(* Logix 5000 project; controller reports 1756-L63 rev 20.15; software revision 20.04; part 20 of 52 *)

        [1198].log_data[8].valid := 1, [1198].log_data[9].valid := 1, [1198].log_data[10].valid := 1, [1198].log_data[11].valid := 1, [1198].log_data[12].valid := 1, [1198].log_data[13].valid := 1, [1198].log_data[14].valid := 1, [1198].log_data[15].valid := 1, [1198].log_data[16].valid := 1, [1198].log_data[17].valid := 1, [1198].log_data[18].valid := 1, [1198].log_data[19].valid := 1, [1198].time.Year := 2023, [1198].time.Month := 1, [1198].time.Day := 13, [1198].time.Hour := 20, [1198].time.Minute := 14, [1198].time.Second := 59, [1199].log_data[0].min := 1.0, [1199].log_data[0].max := 1.0, [1199].log_data[0].total := 300.0, [1199].log_data[0].time := 300.0, [1199].log_data[0].minminute := 15, [1199].log_data[0].maxminute := 15, [1199].log_data[0].valid := 1, [1199].log_data[1].valid := 1, [1199].log_data[2].valid := 1, [1199].log_data[3].valid := 1, [1199].log_data[4].valid := 1, [1199].log_data[5].valid := 1, [1199].log_data[6].valid := 1, [1199].log_data[7].valid := 1, [1199].log_data[8].valid := 1, [1199].log_data[9].valid := 1, [1199].log_data[10].valid := 1, [1199].log_data[11].valid := 1, [1199].log_data[12].valid := 1, [1199].log_data[13].valid := 1, [1199].log_data[14].valid := 1, [1199].log_data[15].valid := 1, [1199].log_data[16].valid := 1, [1199].log_data[17].valid := 1, [1199].log_data[18].valid := 1, [1199].log_data[19].valid := 1, [1199].time.Year := 2023, [1199].time.Month := 1, [1199].time.Day := 13, [1199].time.Hour := 20, [1199].time.Minute := 19, [1199].time.Second := 59, [1200].log_data[0].min := 1.0, [1200].log_data[0].max := 1.0, [1200].log_data[0].total := 300.0, [1200].log_data[0].time := 300.0, [1200].log_data[0].minminute := 20, [1200].log_data[0].maxminute := 20, [1200].log_data[0].valid := 1, [1200].log_data[1].valid := 1, [1200].log_data[2].valid := 1, [1200].log_data[3].valid := 1,
        [1200].log_data[4].valid := 1, [1200].log_data[5].valid := 1, [1200].log_data[6].valid := 1, [1200].log_data[7].valid := 1, [1200].log_data[8].valid := 1, [1200].log_data[9].valid := 1, [1200].log_data[10].valid := 1, [1200].log_data[11].valid := 1, [1200].log_data[12].valid := 1, [1200].log_data[13].valid := 1, [1200].log_data[14].valid := 1, [1200].log_data[15].valid := 1, [1200].log_data[16].valid := 1, [1200].log_data[17].valid := 1, [1200].log_data[18].valid := 1, [1200].log_data[19].valid := 1, [1200].time.Year := 2023, [1200].time.Month := 1, [1200].time.Day := 13, [1200].time.Hour := 20, [1200].time.Minute := 24, [1200].time.Second := 59, [1201].log_data[0].min := 1.0, [1201].log_data[0].max := 1.0, [1201].log_data[0].total := 300.0, [1201].log_data[0].time := 300.0, [1201].log_data[0].minminute := 25, [1201].log_data[0].maxminute := 25, [1201].log_data[0].valid := 1, [1201].log_data[1].valid := 1, [1201].log_data[2].valid := 1, [1201].log_data[3].valid := 1, [1201].log_data[4].valid := 1, [1201].log_data[5].valid := 1, [1201].log_data[6].valid := 1, [1201].log_data[7].valid := 1, [1201].log_data[8].valid := 1, [1201].log_data[9].valid := 1, [1201].log_data[10].valid := 1, [1201].log_data[11].valid := 1, [1201].log_data[12].valid := 1, [1201].log_data[13].valid := 1, [1201].log_data[14].valid := 1, [1201].log_data[15].valid := 1, [1201].log_data[16].valid := 1, [1201].log_data[17].valid := 1, [1201].log_data[18].valid := 1, [1201].log_data[19].valid := 1, [1201].time.Year := 2023, [1201].time.Month := 1, [1201].time.Day := 13, [1201].time.Hour := 20, [1201].time.Minute := 29, [1201].time.Second := 59, [1202].log_data[0].min := 1.0, [1202].log_data[0].max := 1.0, [1202].log_data[0].total := 300.0, [1202].log_data[0].time := 300.0, [1202].log_data[0].minminute := 30, [1202].log_data[0].maxminute := 30,
        [1202].log_data[0].valid := 1, [1202].log_data[1].valid := 1, [1202].log_data[2].valid := 1, [1202].log_data[3].valid := 1, [1202].log_data[4].valid := 1, [1202].log_data[5].valid := 1, [1202].log_data[6].valid := 1, [1202].log_data[7].valid := 1, [1202].log_data[8].valid := 1, [1202].log_data[9].valid := 1, [1202].log_data[10].valid := 1, [1202].log_data[11].valid := 1, [1202].log_data[12].valid := 1, [1202].log_data[13].valid := 1, [1202].log_data[14].valid := 1, [1202].log_data[15].valid := 1, [1202].log_data[16].valid := 1, [1202].log_data[17].valid := 1, [1202].log_data[18].valid := 1, [1202].log_data[19].valid := 1, [1202].time.Year := 2023, [1202].time.Month := 1, [1202].time.Day := 13, [1202].time.Hour := 20, [1202].time.Minute := 34, [1202].time.Second := 59, [1203].log_data[0].min := 1.0, [1203].log_data[0].max := 1.0, [1203].log_data[0].total := 300.0, [1203].log_data[0].time := 300.0, [1203].log_data[0].minminute := 35, [1203].log_data[0].maxminute := 35, [1203].log_data[0].valid := 1, [1203].log_data[1].valid := 1, [1203].log_data[2].valid := 1, [1203].log_data[3].valid := 1, [1203].log_data[4].valid := 1, [1203].log_data[5].valid := 1, [1203].log_data[6].valid := 1, [1203].log_data[7].valid := 1, [1203].log_data[8].valid := 1, [1203].log_data[9].valid := 1, [1203].log_data[10].valid := 1, [1203].log_data[11].valid := 1, [1203].log_data[12].valid := 1, [1203].log_data[13].valid := 1, [1203].log_data[14].valid := 1, [1203].log_data[15].valid := 1, [1203].log_data[16].valid := 1, [1203].log_data[17].valid := 1, [1203].log_data[18].valid := 1, [1203].log_data[19].valid := 1, [1203].time.Year := 2023, [1203].time.Month := 1, [1203].time.Day := 13, [1203].time.Hour := 20, [1203].time.Minute := 39, [1203].time.Second := 59, [1204].log_data[0].min := 1.0, [1204].log_data[0].max := 1.0,
        [1204].log_data[0].total := 300.0, [1204].log_data[0].time := 300.0, [1204].log_data[0].minminute := 40, [1204].log_data[0].maxminute := 40, [1204].log_data[0].valid := 1, [1204].log_data[1].valid := 1, [1204].log_data[2].valid := 1, [1204].log_data[3].valid := 1, [1204].log_data[4].valid := 1, [1204].log_data[5].valid := 1, [1204].log_data[6].valid := 1, [1204].log_data[7].valid := 1, [1204].log_data[8].valid := 1, [1204].log_data[9].valid := 1, [1204].log_data[10].valid := 1, [1204].log_data[11].valid := 1, [1204].log_data[12].valid := 1, [1204].log_data[13].valid := 1, [1204].log_data[14].valid := 1, [1204].log_data[15].valid := 1, [1204].log_data[16].valid := 1, [1204].log_data[17].valid := 1, [1204].log_data[18].valid := 1, [1204].log_data[19].valid := 1, [1204].time.Year := 2023, [1204].time.Month := 1, [1204].time.Day := 13, [1204].time.Hour := 20, [1204].time.Minute := 44, [1204].time.Second := 59, [1205].log_data[0].min := 1.0, [1205].log_data[0].max := 1.0, [1205].log_data[0].total := 300.0, [1205].log_data[0].time := 300.0, [1205].log_data[0].minminute := 45, [1205].log_data[0].maxminute := 45, [1205].log_data[0].valid := 1, [1205].log_data[1].valid := 1, [1205].log_data[2].valid := 1, [1205].log_data[3].valid := 1, [1205].log_data[4].valid := 1, [1205].log_data[5].valid := 1, [1205].log_data[6].valid := 1, [1205].log_data[7].valid := 1, [1205].log_data[8].valid := 1, [1205].log_data[9].valid := 1, [1205].log_data[10].valid := 1, [1205].log_data[11].valid := 1, [1205].log_data[12].valid := 1, [1205].log_data[13].valid := 1, [1205].log_data[14].valid := 1, [1205].log_data[15].valid := 1, [1205].log_data[16].valid := 1, [1205].log_data[17].valid := 1, [1205].log_data[18].valid := 1, [1205].log_data[19].valid := 1, [1205].time.Year := 2023, [1205].time.Month := 1, [1205].time.Day := 13, [1205].time.Hour := 20,
        [1205].time.Minute := 49, [1205].time.Second := 59, [1206].log_data[0].min := 1.0, [1206].log_data[0].max := 1.0, [1206].log_data[0].total := 300.0, [1206].log_data[0].time := 300.0, [1206].log_data[0].minminute := 50, [1206].log_data[0].maxminute := 50, [1206].log_data[0].valid := 1, [1206].log_data[1].valid := 1, [1206].log_data[2].valid := 1, [1206].log_data[3].valid := 1, [1206].log_data[4].valid := 1, [1206].log_data[5].valid := 1, [1206].log_data[6].valid := 1, [1206].log_data[7].valid := 1, [1206].log_data[8].valid := 1, [1206].log_data[9].valid := 1, [1206].log_data[10].valid := 1, [1206].log_data[11].valid := 1, [1206].log_data[12].valid := 1, [1206].log_data[13].valid := 1, [1206].log_data[14].valid := 1, [1206].log_data[15].valid := 1, [1206].log_data[16].valid := 1, [1206].log_data[17].valid := 1, [1206].log_data[18].valid := 1, [1206].log_data[19].valid := 1, [1206].time.Year := 2023, [1206].time.Month := 1, [1206].time.Day := 13, [1206].time.Hour := 20, [1206].time.Minute := 54, [1206].time.Second := 59, [1207].log_data[0].min := 1.0, [1207].log_data[0].max := 1.0, [1207].log_data[0].total := 300.0, [1207].log_data[0].time := 300.0, [1207].log_data[0].minminute := 55, [1207].log_data[0].maxminute := 55, [1207].log_data[0].valid := 1, [1207].log_data[1].valid := 1, [1207].log_data[2].valid := 1, [1207].log_data[3].valid := 1, [1207].log_data[4].valid := 1, [1207].log_data[5].valid := 1, [1207].log_data[6].valid := 1, [1207].log_data[7].valid := 1, [1207].log_data[8].valid := 1, [1207].log_data[9].valid := 1, [1207].log_data[10].valid := 1, [1207].log_data[11].valid := 1, [1207].log_data[12].valid := 1, [1207].log_data[13].valid := 1, [1207].log_data[14].valid := 1, [1207].log_data[15].valid := 1, [1207].log_data[16].valid := 1, [1207].log_data[17].valid := 1, [1207].log_data[18].valid := 1, [1207].log_data[19].valid := 1,
        [1207].time.Year := 2023, [1207].time.Month := 1, [1207].time.Day := 13, [1207].time.Hour := 20, [1207].time.Minute := 59, [1207].time.Second := 59, [1208].log_data[0].min := 1.0, [1208].log_data[0].max := 1.0, [1208].log_data[0].total := 300.0, [1208].log_data[0].time := 300.0, [1208].log_data[0].valid := 1, [1208].log_data[1].valid := 1, [1208].log_data[2].valid := 1, [1208].log_data[3].valid := 1, [1208].log_data[4].valid := 1, [1208].log_data[5].valid := 1, [1208].log_data[6].valid := 1, [1208].log_data[7].valid := 1, [1208].log_data[8].valid := 1, [1208].log_data[9].valid := 1, [1208].log_data[10].valid := 1, [1208].log_data[11].valid := 1, [1208].log_data[12].valid := 1, [1208].log_data[13].valid := 1, [1208].log_data[14].valid := 1, [1208].log_data[15].valid := 1, [1208].log_data[16].valid := 1, [1208].log_data[17].valid := 1, [1208].log_data[18].valid := 1, [1208].log_data[19].valid := 1, [1208].time.Year := 2023, [1208].time.Month := 1, [1208].time.Day := 13, [1208].time.Hour := 21, [1208].time.Minute := 4, [1208].time.Second := 59, [1209].log_data[0].min := 1.0, [1209].log_data[0].max := 1.0, [1209].log_data[0].total := 300.0, [1209].log_data[0].time := 300.0, [1209].log_data[0].minminute := 5, [1209].log_data[0].maxminute := 5, [1209].log_data[0].valid := 1, [1209].log_data[1].valid := 1, [1209].log_data[2].valid := 1, [1209].log_data[3].valid := 1, [1209].log_data[4].valid := 1, [1209].log_data[5].valid := 1, [1209].log_data[6].valid := 1, [1209].log_data[7].valid := 1, [1209].log_data[8].valid := 1, [1209].log_data[9].valid := 1, [1209].log_data[10].valid := 1, [1209].log_data[11].valid := 1, [1209].log_data[12].valid := 1, [1209].log_data[13].valid := 1, [1209].log_data[14].valid := 1, [1209].log_data[15].valid := 1, [1209].log_data[16].valid := 1, [1209].log_data[17].valid := 1,
        [1209].log_data[18].valid := 1, [1209].log_data[19].valid := 1, [1209].time.Year := 2023, [1209].time.Month := 1, [1209].time.Day := 13, [1209].time.Hour := 21, [1209].time.Minute := 9, [1209].time.Second := 59, [1210].log_data[0].min := 1.0, [1210].log_data[0].max := 1.0, [1210].log_data[0].total := 300.0, [1210].log_data[0].time := 300.0, [1210].log_data[0].minminute := 10, [1210].log_data[0].maxminute := 10, [1210].log_data[0].valid := 1, [1210].log_data[1].valid := 1, [1210].log_data[2].valid := 1, [1210].log_data[3].valid := 1, [1210].log_data[4].valid := 1, [1210].log_data[5].valid := 1, [1210].log_data[6].valid := 1, [1210].log_data[7].valid := 1, [1210].log_data[8].valid := 1, [1210].log_data[9].valid := 1, [1210].log_data[10].valid := 1, [1210].log_data[11].valid := 1, [1210].log_data[12].valid := 1, [1210].log_data[13].valid := 1, [1210].log_data[14].valid := 1, [1210].log_data[15].valid := 1, [1210].log_data[16].valid := 1, [1210].log_data[17].valid := 1, [1210].log_data[18].valid := 1, [1210].log_data[19].valid := 1, [1210].time.Year := 2023, [1210].time.Month := 1, [1210].time.Day := 13, [1210].time.Hour := 21, [1210].time.Minute := 14, [1210].time.Second := 59, [1211].log_data[0].min := 1.0, [1211].log_data[0].max := 1.0, [1211].log_data[0].total := 300.0, [1211].log_data[0].time := 300.0, [1211].log_data[0].minminute := 15, [1211].log_data[0].maxminute := 15, [1211].log_data[0].valid := 1, [1211].log_data[1].valid := 1, [1211].log_data[2].valid := 1, [1211].log_data[3].valid := 1, [1211].log_data[4].valid := 1, [1211].log_data[5].valid := 1, [1211].log_data[6].valid := 1, [1211].log_data[7].valid := 1, [1211].log_data[8].valid := 1, [1211].log_data[9].valid := 1, [1211].log_data[10].valid := 1, [1211].log_data[11].valid := 1, [1211].log_data[12].valid := 1, [1211].log_data[13].valid := 1,
        [1211].log_data[14].valid := 1, [1211].log_data[15].valid := 1, [1211].log_data[16].valid := 1, [1211].log_data[17].valid := 1, [1211].log_data[18].valid := 1, [1211].log_data[19].valid := 1, [1211].time.Year := 2023, [1211].time.Month := 1, [1211].time.Day := 13, [1211].time.Hour := 21, [1211].time.Minute := 19, [1211].time.Second := 59, [1212].log_data[0].min := 1.0, [1212].log_data[0].max := 1.0, [1212].log_data[0].total := 300.0, [1212].log_data[0].time := 300.0, [1212].log_data[0].minminute := 20, [1212].log_data[0].maxminute := 20, [1212].log_data[0].valid := 1, [1212].log_data[1].valid := 1, [1212].log_data[2].valid := 1, [1212].log_data[3].valid := 1, [1212].log_data[4].valid := 1, [1212].log_data[5].valid := 1, [1212].log_data[6].valid := 1, [1212].log_data[7].valid := 1, [1212].log_data[8].valid := 1, [1212].log_data[9].valid := 1, [1212].log_data[10].valid := 1, [1212].log_data[11].valid := 1, [1212].log_data[12].valid := 1, [1212].log_data[13].valid := 1, [1212].log_data[14].valid := 1, [1212].log_data[15].valid := 1, [1212].log_data[16].valid := 1, [1212].log_data[17].valid := 1, [1212].log_data[18].valid := 1, [1212].log_data[19].valid := 1, [1212].time.Year := 2023, [1212].time.Month := 1, [1212].time.Day := 13, [1212].time.Hour := 21, [1212].time.Minute := 24, [1212].time.Second := 59, [1213].log_data[0].min := 1.0, [1213].log_data[0].max := 1.0, [1213].log_data[0].total := 300.0, [1213].log_data[0].time := 300.0, [1213].log_data[0].minminute := 25, [1213].log_data[0].maxminute := 25, [1213].log_data[0].valid := 1, [1213].log_data[1].valid := 1, [1213].log_data[2].valid := 1, [1213].log_data[3].valid := 1, [1213].log_data[4].valid := 1, [1213].log_data[5].valid := 1, [1213].log_data[6].valid := 1, [1213].log_data[7].valid := 1, [1213].log_data[8].valid := 1, [1213].log_data[9].valid := 1,
        [1213].log_data[10].valid := 1, [1213].log_data[11].valid := 1, [1213].log_data[12].valid := 1, [1213].log_data[13].valid := 1, [1213].log_data[14].valid := 1, [1213].log_data[15].valid := 1, [1213].log_data[16].valid := 1, [1213].log_data[17].valid := 1, [1213].log_data[18].valid := 1, [1213].log_data[19].valid := 1, [1213].time.Year := 2023, [1213].time.Month := 1, [1213].time.Day := 13, [1213].time.Hour := 21, [1213].time.Minute := 29, [1213].time.Second := 59, [1214].log_data[0].min := 1.0, [1214].log_data[0].max := 1.0, [1214].log_data[0].total := 300.0, [1214].log_data[0].time := 300.0, [1214].log_data[0].minminute := 30, [1214].log_data[0].maxminute := 30, [1214].log_data[0].valid := 1, [1214].log_data[1].valid := 1, [1214].log_data[2].valid := 1, [1214].log_data[3].valid := 1, [1214].log_data[4].valid := 1, [1214].log_data[5].valid := 1, [1214].log_data[6].valid := 1, [1214].log_data[7].valid := 1, [1214].log_data[8].valid := 1, [1214].log_data[9].valid := 1, [1214].log_data[10].valid := 1, [1214].log_data[11].valid := 1, [1214].log_data[12].valid := 1, [1214].log_data[13].valid := 1, [1214].log_data[14].valid := 1, [1214].log_data[15].valid := 1, [1214].log_data[16].valid := 1, [1214].log_data[17].valid := 1, [1214].log_data[18].valid := 1, [1214].log_data[19].valid := 1, [1214].time.Year := 2023, [1214].time.Month := 1, [1214].time.Day := 13, [1214].time.Hour := 21, [1214].time.Minute := 34, [1214].time.Second := 59, [1215].log_data[0].min := 1.0, [1215].log_data[0].max := 1.0, [1215].log_data[0].total := 300.0, [1215].log_data[0].time := 300.0, [1215].log_data[0].minminute := 35, [1215].log_data[0].maxminute := 35, [1215].log_data[0].valid := 1, [1215].log_data[1].valid := 1, [1215].log_data[2].valid := 1, [1215].log_data[3].valid := 1, [1215].log_data[4].valid := 1, [1215].log_data[5].valid := 1,
        [1215].log_data[6].valid := 1, [1215].log_data[7].valid := 1, [1215].log_data[8].valid := 1, [1215].log_data[9].valid := 1, [1215].log_data[10].valid := 1, [1215].log_data[11].valid := 1, [1215].log_data[12].valid := 1, [1215].log_data[13].valid := 1, [1215].log_data[14].valid := 1, [1215].log_data[15].valid := 1, [1215].log_data[16].valid := 1, [1215].log_data[17].valid := 1, [1215].log_data[18].valid := 1, [1215].log_data[19].valid := 1, [1215].time.Year := 2023, [1215].time.Month := 1, [1215].time.Day := 13, [1215].time.Hour := 21, [1215].time.Minute := 39, [1215].time.Second := 59, [1216].log_data[0].min := 1.0, [1216].log_data[0].max := 1.0, [1216].log_data[0].total := 300.0, [1216].log_data[0].time := 300.0, [1216].log_data[0].minminute := 40, [1216].log_data[0].maxminute := 40, [1216].log_data[0].valid := 1, [1216].log_data[1].valid := 1, [1216].log_data[2].valid := 1, [1216].log_data[3].valid := 1, [1216].log_data[4].valid := 1, [1216].log_data[5].valid := 1, [1216].log_data[6].valid := 1, [1216].log_data[7].valid := 1, [1216].log_data[8].valid := 1, [1216].log_data[9].valid := 1, [1216].log_data[10].valid := 1, [1216].log_data[11].valid := 1, [1216].log_data[12].valid := 1, [1216].log_data[13].valid := 1, [1216].log_data[14].valid := 1, [1216].log_data[15].valid := 1, [1216].log_data[16].valid := 1, [1216].log_data[17].valid := 1, [1216].log_data[18].valid := 1, [1216].log_data[19].valid := 1, [1216].time.Year := 2023, [1216].time.Month := 1, [1216].time.Day := 13, [1216].time.Hour := 21, [1216].time.Minute := 44, [1216].time.Second := 59, [1217].log_data[0].min := 1.0, [1217].log_data[0].max := 1.0, [1217].log_data[0].total := 300.0, [1217].log_data[0].time := 300.0, [1217].log_data[0].minminute := 45, [1217].log_data[0].maxminute := 45, [1217].log_data[0].valid := 1, [1217].log_data[1].valid := 1,
        [1217].log_data[2].valid := 1, [1217].log_data[3].valid := 1, [1217].log_data[4].valid := 1, [1217].log_data[5].valid := 1, [1217].log_data[6].valid := 1, [1217].log_data[7].valid := 1, [1217].log_data[8].valid := 1, [1217].log_data[9].valid := 1, [1217].log_data[10].valid := 1, [1217].log_data[11].valid := 1, [1217].log_data[12].valid := 1, [1217].log_data[13].valid := 1, [1217].log_data[14].valid := 1, [1217].log_data[15].valid := 1, [1217].log_data[16].valid := 1, [1217].log_data[17].valid := 1, [1217].log_data[18].valid := 1, [1217].log_data[19].valid := 1, [1217].time.Year := 2023, [1217].time.Month := 1, [1217].time.Day := 13, [1217].time.Hour := 21, [1217].time.Minute := 49, [1217].time.Second := 59, [1218].log_data[0].min := 1.0, [1218].log_data[0].max := 1.0, [1218].log_data[0].total := 300.0, [1218].log_data[0].time := 300.0, [1218].log_data[0].minminute := 50, [1218].log_data[0].maxminute := 50, [1218].log_data[0].valid := 1, [1218].log_data[1].valid := 1, [1218].log_data[2].valid := 1, [1218].log_data[3].valid := 1, [1218].log_data[4].valid := 1, [1218].log_data[5].valid := 1, [1218].log_data[6].valid := 1, [1218].log_data[7].valid := 1, [1218].log_data[8].valid := 1, [1218].log_data[9].valid := 1, [1218].log_data[10].valid := 1, [1218].log_data[11].valid := 1, [1218].log_data[12].valid := 1, [1218].log_data[13].valid := 1, [1218].log_data[14].valid := 1, [1218].log_data[15].valid := 1, [1218].log_data[16].valid := 1, [1218].log_data[17].valid := 1, [1218].log_data[18].valid := 1, [1218].log_data[19].valid := 1, [1218].time.Year := 2023, [1218].time.Month := 1, [1218].time.Day := 13, [1218].time.Hour := 21, [1218].time.Minute := 54, [1218].time.Second := 59, [1219].log_data[0].min := 1.0, [1219].log_data[0].max := 1.0, [1219].log_data[0].total := 300.0, [1219].log_data[0].time := 300.0,
        [1219].log_data[0].minminute := 55, [1219].log_data[0].maxminute := 55, [1219].log_data[0].valid := 1, [1219].log_data[1].valid := 1, [1219].log_data[2].valid := 1, [1219].log_data[3].valid := 1, [1219].log_data[4].valid := 1, [1219].log_data[5].valid := 1, [1219].log_data[6].valid := 1, [1219].log_data[7].valid := 1, [1219].log_data[8].valid := 1, [1219].log_data[9].valid := 1, [1219].log_data[10].valid := 1, [1219].log_data[11].valid := 1, [1219].log_data[12].valid := 1, [1219].log_data[13].valid := 1, [1219].log_data[14].valid := 1, [1219].log_data[15].valid := 1, [1219].log_data[16].valid := 1, [1219].log_data[17].valid := 1, [1219].log_data[18].valid := 1, [1219].log_data[19].valid := 1, [1219].time.Year := 2023, [1219].time.Month := 1, [1219].time.Day := 13, [1219].time.Hour := 21, [1219].time.Minute := 59, [1219].time.Second := 59, [1220].log_data[0].min := 1.0, [1220].log_data[0].max := 1.0, [1220].log_data[0].total := 300.0, [1220].log_data[0].time := 300.0, [1220].log_data[0].valid := 1, [1220].log_data[1].valid := 1, [1220].log_data[2].valid := 1, [1220].log_data[3].valid := 1, [1220].log_data[4].valid := 1, [1220].log_data[5].valid := 1, [1220].log_data[6].valid := 1, [1220].log_data[7].valid := 1, [1220].log_data[8].valid := 1, [1220].log_data[9].valid := 1, [1220].log_data[10].valid := 1, [1220].log_data[11].valid := 1, [1220].log_data[12].valid := 1, [1220].log_data[13].valid := 1, [1220].log_data[14].valid := 1, [1220].log_data[15].valid := 1, [1220].log_data[16].valid := 1, [1220].log_data[17].valid := 1, [1220].log_data[18].valid := 1, [1220].log_data[19].valid := 1, [1220].time.Year := 2023, [1220].time.Month := 1, [1220].time.Day := 13, [1220].time.Hour := 22, [1220].time.Minute := 4, [1220].time.Second := 59, [1221].log_data[0].min := 1.0, [1221].log_data[0].max := 1.0,
        [1221].log_data[0].total := 300.0, [1221].log_data[0].time := 300.0, [1221].log_data[0].minminute := 5, [1221].log_data[0].maxminute := 5, [1221].log_data[0].valid := 1, [1221].log_data[1].valid := 1, [1221].log_data[2].valid := 1, [1221].log_data[3].valid := 1, [1221].log_data[4].valid := 1, [1221].log_data[5].valid := 1, [1221].log_data[6].valid := 1, [1221].log_data[7].valid := 1, [1221].log_data[8].valid := 1, [1221].log_data[9].valid := 1, [1221].log_data[10].valid := 1, [1221].log_data[11].valid := 1, [1221].log_data[12].valid := 1, [1221].log_data[13].valid := 1, [1221].log_data[14].valid := 1, [1221].log_data[15].valid := 1, [1221].log_data[16].valid := 1, [1221].log_data[17].valid := 1, [1221].log_data[18].valid := 1, [1221].log_data[19].valid := 1, [1221].time.Year := 2023, [1221].time.Month := 1, [1221].time.Day := 13, [1221].time.Hour := 22, [1221].time.Minute := 9, [1221].time.Second := 59, [1222].log_data[0].min := 1.0, [1222].log_data[0].max := 1.0, [1222].log_data[0].total := 300.0, [1222].log_data[0].time := 300.0, [1222].log_data[0].minminute := 10, [1222].log_data[0].maxminute := 10, [1222].log_data[0].valid := 1, [1222].log_data[1].valid := 1, [1222].log_data[2].valid := 1, [1222].log_data[3].valid := 1, [1222].log_data[4].valid := 1, [1222].log_data[5].valid := 1, [1222].log_data[6].valid := 1, [1222].log_data[7].valid := 1, [1222].log_data[8].valid := 1, [1222].log_data[9].valid := 1, [1222].log_data[10].valid := 1, [1222].log_data[11].valid := 1, [1222].log_data[12].valid := 1, [1222].log_data[13].valid := 1, [1222].log_data[14].valid := 1, [1222].log_data[15].valid := 1, [1222].log_data[16].valid := 1, [1222].log_data[17].valid := 1, [1222].log_data[18].valid := 1, [1222].log_data[19].valid := 1, [1222].time.Year := 2023, [1222].time.Month := 1, [1222].time.Day := 13, [1222].time.Hour := 22,
        [1222].time.Minute := 14, [1222].time.Second := 59, [1223].log_data[0].min := 1.0, [1223].log_data[0].max := 1.0, [1223].log_data[0].total := 300.0, [1223].log_data[0].time := 300.0, [1223].log_data[0].minminute := 15, [1223].log_data[0].maxminute := 15, [1223].log_data[0].valid := 1, [1223].log_data[1].valid := 1, [1223].log_data[2].valid := 1, [1223].log_data[3].valid := 1, [1223].log_data[4].valid := 1, [1223].log_data[5].valid := 1, [1223].log_data[6].valid := 1, [1223].log_data[7].valid := 1, [1223].log_data[8].valid := 1, [1223].log_data[9].valid := 1, [1223].log_data[10].valid := 1, [1223].log_data[11].valid := 1, [1223].log_data[12].valid := 1, [1223].log_data[13].valid := 1, [1223].log_data[14].valid := 1, [1223].log_data[15].valid := 1, [1223].log_data[16].valid := 1, [1223].log_data[17].valid := 1, [1223].log_data[18].valid := 1, [1223].log_data[19].valid := 1, [1223].time.Year := 2023, [1223].time.Month := 1, [1223].time.Day := 13, [1223].time.Hour := 22, [1223].time.Minute := 19, [1223].time.Second := 59, [1224].log_data[0].min := 1.0, [1224].log_data[0].max := 1.0, [1224].log_data[0].total := 300.0, [1224].log_data[0].time := 300.0, [1224].log_data[0].minminute := 20, [1224].log_data[0].maxminute := 20, [1224].log_data[0].valid := 1, [1224].log_data[1].valid := 1, [1224].log_data[2].valid := 1, [1224].log_data[3].valid := 1, [1224].log_data[4].valid := 1, [1224].log_data[5].valid := 1, [1224].log_data[6].valid := 1, [1224].log_data[7].valid := 1, [1224].log_data[8].valid := 1, [1224].log_data[9].valid := 1, [1224].log_data[10].valid := 1, [1224].log_data[11].valid := 1, [1224].log_data[12].valid := 1, [1224].log_data[13].valid := 1, [1224].log_data[14].valid := 1, [1224].log_data[15].valid := 1, [1224].log_data[16].valid := 1, [1224].log_data[17].valid := 1, [1224].log_data[18].valid := 1, [1224].log_data[19].valid := 1,
        [1224].time.Year := 2023, [1224].time.Month := 1, [1224].time.Day := 13, [1224].time.Hour := 22, [1224].time.Minute := 24, [1224].time.Second := 59, [1225].log_data[0].min := 1.0, [1225].log_data[0].max := 1.0, [1225].log_data[0].total := 300.0, [1225].log_data[0].time := 300.0, [1225].log_data[0].minminute := 25, [1225].log_data[0].maxminute := 25, [1225].log_data[0].valid := 1, [1225].log_data[1].valid := 1, [1225].log_data[2].valid := 1, [1225].log_data[3].valid := 1, [1225].log_data[4].valid := 1, [1225].log_data[5].valid := 1, [1225].log_data[6].valid := 1, [1225].log_data[7].valid := 1, [1225].log_data[8].valid := 1, [1225].log_data[9].valid := 1, [1225].log_data[10].valid := 1, [1225].log_data[11].valid := 1, [1225].log_data[12].valid := 1, [1225].log_data[13].valid := 1, [1225].log_data[14].valid := 1, [1225].log_data[15].valid := 1, [1225].log_data[16].valid := 1, [1225].log_data[17].valid := 1, [1225].log_data[18].valid := 1, [1225].log_data[19].valid := 1, [1225].time.Year := 2023, [1225].time.Month := 1, [1225].time.Day := 13, [1225].time.Hour := 22, [1225].time.Minute := 29, [1225].time.Second := 59, [1226].log_data[0].min := 1.0, [1226].log_data[0].max := 1.0, [1226].log_data[0].total := 300.0, [1226].log_data[0].time := 300.0, [1226].log_data[0].minminute := 30, [1226].log_data[0].maxminute := 30, [1226].log_data[0].valid := 1, [1226].log_data[1].valid := 1, [1226].log_data[2].valid := 1, [1226].log_data[3].valid := 1, [1226].log_data[4].valid := 1, [1226].log_data[5].valid := 1, [1226].log_data[6].valid := 1, [1226].log_data[7].valid := 1, [1226].log_data[8].valid := 1, [1226].log_data[9].valid := 1, [1226].log_data[10].valid := 1, [1226].log_data[11].valid := 1, [1226].log_data[12].valid := 1, [1226].log_data[13].valid := 1, [1226].log_data[14].valid := 1, [1226].log_data[15].valid := 1,
        [1226].log_data[16].valid := 1, [1226].log_data[17].valid := 1, [1226].log_data[18].valid := 1, [1226].log_data[19].valid := 1, [1226].time.Year := 2023, [1226].time.Month := 1, [1226].time.Day := 13, [1226].time.Hour := 22, [1226].time.Minute := 34, [1226].time.Second := 59, [1227].log_data[0].min := 1.0, [1227].log_data[0].max := 1.0, [1227].log_data[0].total := 300.0, [1227].log_data[0].time := 300.0, [1227].log_data[0].minminute := 35, [1227].log_data[0].maxminute := 35, [1227].log_data[0].valid := 1, [1227].log_data[1].valid := 1, [1227].log_data[2].valid := 1, [1227].log_data[3].valid := 1, [1227].log_data[4].valid := 1, [1227].log_data[5].valid := 1, [1227].log_data[6].valid := 1, [1227].log_data[7].valid := 1, [1227].log_data[8].valid := 1, [1227].log_data[9].valid := 1, [1227].log_data[10].valid := 1, [1227].log_data[11].valid := 1, [1227].log_data[12].valid := 1, [1227].log_data[13].valid := 1, [1227].log_data[14].valid := 1, [1227].log_data[15].valid := 1, [1227].log_data[16].valid := 1, [1227].log_data[17].valid := 1, [1227].log_data[18].valid := 1, [1227].log_data[19].valid := 1, [1227].time.Year := 2023, [1227].time.Month := 1, [1227].time.Day := 13, [1227].time.Hour := 22, [1227].time.Minute := 39, [1227].time.Second := 59, [1228].log_data[0].min := 1.0, [1228].log_data[0].max := 1.0, [1228].log_data[0].total := 300.0, [1228].log_data[0].time := 300.0, [1228].log_data[0].minminute := 40, [1228].log_data[0].maxminute := 40, [1228].log_data[0].valid := 1, [1228].log_data[1].valid := 1, [1228].log_data[2].valid := 1, [1228].log_data[3].valid := 1, [1228].log_data[4].valid := 1, [1228].log_data[5].valid := 1, [1228].log_data[6].valid := 1, [1228].log_data[7].valid := 1, [1228].log_data[8].valid := 1, [1228].log_data[9].valid := 1, [1228].log_data[10].valid := 1, [1228].log_data[11].valid := 1,
        [1228].log_data[12].valid := 1, [1228].log_data[13].valid := 1, [1228].log_data[14].valid := 1, [1228].log_data[15].valid := 1, [1228].log_data[16].valid := 1, [1228].log_data[17].valid := 1, [1228].log_data[18].valid := 1, [1228].log_data[19].valid := 1, [1228].time.Year := 2023, [1228].time.Month := 1, [1228].time.Day := 13, [1228].time.Hour := 22, [1228].time.Minute := 44, [1228].time.Second := 59, [1229].log_data[0].min := 1.0, [1229].log_data[0].max := 1.0, [1229].log_data[0].total := 300.0, [1229].log_data[0].time := 300.0, [1229].log_data[0].minminute := 45, [1229].log_data[0].maxminute := 45, [1229].log_data[0].valid := 1, [1229].log_data[1].valid := 1, [1229].log_data[2].valid := 1, [1229].log_data[3].valid := 1, [1229].log_data[4].valid := 1, [1229].log_data[5].valid := 1, [1229].log_data[6].valid := 1, [1229].log_data[7].valid := 1, [1229].log_data[8].valid := 1, [1229].log_data[9].valid := 1, [1229].log_data[10].valid := 1, [1229].log_data[11].valid := 1, [1229].log_data[12].valid := 1, [1229].log_data[13].valid := 1, [1229].log_data[14].valid := 1, [1229].log_data[15].valid := 1, [1229].log_data[16].valid := 1, [1229].log_data[17].valid := 1, [1229].log_data[18].valid := 1, [1229].log_data[19].valid := 1, [1229].time.Year := 2023, [1229].time.Month := 1, [1229].time.Day := 13, [1229].time.Hour := 22, [1229].time.Minute := 49, [1229].time.Second := 59, [1230].log_data[0].min := 1.0, [1230].log_data[0].max := 1.0, [1230].log_data[0].total := 300.0, [1230].log_data[0].time := 300.0, [1230].log_data[0].minminute := 50, [1230].log_data[0].maxminute := 50, [1230].log_data[0].valid := 1, [1230].log_data[1].valid := 1, [1230].log_data[2].valid := 1, [1230].log_data[3].valid := 1, [1230].log_data[4].valid := 1, [1230].log_data[5].valid := 1, [1230].log_data[6].valid := 1, [1230].log_data[7].valid := 1,
        [1230].log_data[8].valid := 1, [1230].log_data[9].valid := 1, [1230].log_data[10].valid := 1, [1230].log_data[11].valid := 1, [1230].log_data[12].valid := 1, [1230].log_data[13].valid := 1, [1230].log_data[14].valid := 1, [1230].log_data[15].valid := 1, [1230].log_data[16].valid := 1, [1230].log_data[17].valid := 1, [1230].log_data[18].valid := 1, [1230].log_data[19].valid := 1, [1230].time.Year := 2023, [1230].time.Month := 1, [1230].time.Day := 13, [1230].time.Hour := 22, [1230].time.Minute := 54, [1230].time.Second := 59, [1231].log_data[0].min := 1.0, [1231].log_data[0].max := 1.0, [1231].log_data[0].total := 300.0, [1231].log_data[0].time := 300.0, [1231].log_data[0].minminute := 55, [1231].log_data[0].maxminute := 55, [1231].log_data[0].valid := 1, [1231].log_data[1].valid := 1, [1231].log_data[2].valid := 1, [1231].log_data[3].valid := 1, [1231].log_data[4].valid := 1, [1231].log_data[5].valid := 1, [1231].log_data[6].valid := 1, [1231].log_data[7].valid := 1, [1231].log_data[8].valid := 1, [1231].log_data[9].valid := 1, [1231].log_data[10].valid := 1, [1231].log_data[11].valid := 1, [1231].log_data[12].valid := 1, [1231].log_data[13].valid := 1, [1231].log_data[14].valid := 1, [1231].log_data[15].valid := 1, [1231].log_data[16].valid := 1, [1231].log_data[17].valid := 1, [1231].log_data[18].valid := 1, [1231].log_data[19].valid := 1, [1231].time.Year := 2023, [1231].time.Month := 1, [1231].time.Day := 13, [1231].time.Hour := 22, [1231].time.Minute := 59, [1231].time.Second := 59, [1232].log_data[0].min := 1.0, [1232].log_data[0].max := 1.0, [1232].log_data[0].total := 300.0, [1232].log_data[0].time := 300.0, [1232].log_data[0].valid := 1, [1232].log_data[1].valid := 1, [1232].log_data[2].valid := 1, [1232].log_data[3].valid := 1, [1232].log_data[4].valid := 1, [1232].log_data[5].valid := 1,
        [1232].log_data[6].valid := 1, [1232].log_data[7].valid := 1, [1232].log_data[8].valid := 1, [1232].log_data[9].valid := 1, [1232].log_data[10].valid := 1, [1232].log_data[11].valid := 1, [1232].log_data[12].valid := 1, [1232].log_data[13].valid := 1, [1232].log_data[14].valid := 1, [1232].log_data[15].valid := 1, [1232].log_data[16].valid := 1, [1232].log_data[17].valid := 1, [1232].log_data[18].valid := 1, [1232].log_data[19].valid := 1, [1232].time.Year := 2023, [1232].time.Month := 1, [1232].time.Day := 13, [1232].time.Hour := 23, [1232].time.Minute := 4, [1232].time.Second := 59, [1233].log_data[0].min := 1.0, [1233].log_data[0].max := 1.0, [1233].log_data[0].total := 300.0, [1233].log_data[0].time := 300.0, [1233].log_data[0].minminute := 5, [1233].log_data[0].maxminute := 5, [1233].log_data[0].valid := 1, [1233].log_data[1].valid := 1, [1233].log_data[2].valid := 1, [1233].log_data[3].valid := 1, [1233].log_data[4].valid := 1, [1233].log_data[5].valid := 1, [1233].log_data[6].valid := 1, [1233].log_data[7].valid := 1, [1233].log_data[8].valid := 1, [1233].log_data[9].valid := 1, [1233].log_data[10].valid := 1, [1233].log_data[11].valid := 1, [1233].log_data[12].valid := 1, [1233].log_data[13].valid := 1, [1233].log_data[14].valid := 1, [1233].log_data[15].valid := 1, [1233].log_data[16].valid := 1, [1233].log_data[17].valid := 1, [1233].log_data[18].valid := 1, [1233].log_data[19].valid := 1, [1233].time.Year := 2023, [1233].time.Month := 1, [1233].time.Day := 13, [1233].time.Hour := 23, [1233].time.Minute := 9, [1233].time.Second := 59, [1234].log_data[0].min := 1.0, [1234].log_data[0].max := 1.0, [1234].log_data[0].total := 300.0, [1234].log_data[0].time := 300.0, [1234].log_data[0].minminute := 10, [1234].log_data[0].maxminute := 10, [1234].log_data[0].valid := 1, [1234].log_data[1].valid := 1,
        [1234].log_data[2].valid := 1, [1234].log_data[3].valid := 1, [1234].log_data[4].valid := 1, [1234].log_data[5].valid := 1, [1234].log_data[6].valid := 1, [1234].log_data[7].valid := 1, [1234].log_data[8].valid := 1, [1234].log_data[9].valid := 1, [1234].log_data[10].valid := 1, [1234].log_data[11].valid := 1, [1234].log_data[12].valid := 1, [1234].log_data[13].valid := 1, [1234].log_data[14].valid := 1, [1234].log_data[15].valid := 1, [1234].log_data[16].valid := 1, [1234].log_data[17].valid := 1, [1234].log_data[18].valid := 1, [1234].log_data[19].valid := 1, [1234].time.Year := 2023, [1234].time.Month := 1, [1234].time.Day := 13, [1234].time.Hour := 23, [1234].time.Minute := 14, [1234].time.Second := 59, [1235].log_data[0].min := 1.0, [1235].log_data[0].max := 1.0, [1235].log_data[0].total := 300.0, [1235].log_data[0].time := 300.0, [1235].log_data[0].minminute := 15, [1235].log_data[0].maxminute := 15, [1235].log_data[0].valid := 1, [1235].log_data[1].valid := 1, [1235].log_data[2].valid := 1, [1235].log_data[3].valid := 1, [1235].log_data[4].valid := 1, [1235].log_data[5].valid := 1, [1235].log_data[6].valid := 1, [1235].log_data[7].valid := 1, [1235].log_data[8].valid := 1, [1235].log_data[9].valid := 1, [1235].log_data[10].valid := 1, [1235].log_data[11].valid := 1, [1235].log_data[12].valid := 1, [1235].log_data[13].valid := 1, [1235].log_data[14].valid := 1, [1235].log_data[15].valid := 1, [1235].log_data[16].valid := 1, [1235].log_data[17].valid := 1, [1235].log_data[18].valid := 1, [1235].log_data[19].valid := 1, [1235].time.Year := 2023, [1235].time.Month := 1, [1235].time.Day := 13, [1235].time.Hour := 23, [1235].time.Minute := 19, [1235].time.Second := 59, [1236].log_data[0].min := 1.0, [1236].log_data[0].max := 1.0, [1236].log_data[0].total := 300.0, [1236].log_data[0].time := 300.0,
        [1236].log_data[0].minminute := 20, [1236].log_data[0].maxminute := 20, [1236].log_data[0].valid := 1, [1236].log_data[1].valid := 1, [1236].log_data[2].valid := 1, [1236].log_data[3].valid := 1, [1236].log_data[4].valid := 1, [1236].log_data[5].valid := 1, [1236].log_data[6].valid := 1, [1236].log_data[7].valid := 1, [1236].log_data[8].valid := 1, [1236].log_data[9].valid := 1, [1236].log_data[10].valid := 1, [1236].log_data[11].valid := 1, [1236].log_data[12].valid := 1, [1236].log_data[13].valid := 1, [1236].log_data[14].valid := 1, [1236].log_data[15].valid := 1, [1236].log_data[16].valid := 1, [1236].log_data[17].valid := 1, [1236].log_data[18].valid := 1, [1236].log_data[19].valid := 1, [1236].time.Year := 2023, [1236].time.Month := 1, [1236].time.Day := 13, [1236].time.Hour := 23, [1236].time.Minute := 24, [1236].time.Second := 59, [1237].log_data[0].min := 1.0, [1237].log_data[0].max := 1.0, [1237].log_data[0].total := 300.0, [1237].log_data[0].time := 300.0, [1237].log_data[0].minminute := 25, [1237].log_data[0].maxminute := 25, [1237].log_data[0].valid := 1, [1237].log_data[1].valid := 1, [1237].log_data[2].valid := 1, [1237].log_data[3].valid := 1, [1237].log_data[4].valid := 1, [1237].log_data[5].valid := 1, [1237].log_data[6].valid := 1, [1237].log_data[7].valid := 1, [1237].log_data[8].valid := 1, [1237].log_data[9].valid := 1, [1237].log_data[10].valid := 1, [1237].log_data[11].valid := 1, [1237].log_data[12].valid := 1, [1237].log_data[13].valid := 1, [1237].log_data[14].valid := 1, [1237].log_data[15].valid := 1, [1237].log_data[16].valid := 1, [1237].log_data[17].valid := 1, [1237].log_data[18].valid := 1, [1237].log_data[19].valid := 1, [1237].time.Year := 2023, [1237].time.Month := 1, [1237].time.Day := 13, [1237].time.Hour := 23, [1237].time.Minute := 29, [1237].time.Second := 59,
        [1238].log_data[0].min := 1.0, [1238].log_data[0].max := 1.0, [1238].log_data[0].total := 300.0, [1238].log_data[0].time := 300.0, [1238].log_data[0].minminute := 30, [1238].log_data[0].maxminute := 30, [1238].log_data[0].valid := 1, [1238].log_data[1].valid := 1, [1238].log_data[2].valid := 1, [1238].log_data[3].valid := 1, [1238].log_data[4].valid := 1, [1238].log_data[5].valid := 1, [1238].log_data[6].valid := 1, [1238].log_data[7].valid := 1, [1238].log_data[8].valid := 1, [1238].log_data[9].valid := 1, [1238].log_data[10].valid := 1, [1238].log_data[11].valid := 1, [1238].log_data[12].valid := 1, [1238].log_data[13].valid := 1, [1238].log_data[14].valid := 1, [1238].log_data[15].valid := 1, [1238].log_data[16].valid := 1, [1238].log_data[17].valid := 1, [1238].log_data[18].valid := 1, [1238].log_data[19].valid := 1, [1238].time.Year := 2023, [1238].time.Month := 1, [1238].time.Day := 13, [1238].time.Hour := 23, [1238].time.Minute := 34, [1238].time.Second := 59, [1239].log_data[0].min := 1.0, [1239].log_data[0].max := 1.0, [1239].log_data[0].total := 300.0, [1239].log_data[0].time := 300.0, [1239].log_data[0].minminute := 35, [1239].log_data[0].maxminute := 35, [1239].log_data[0].valid := 1, [1239].log_data[1].valid := 1, [1239].log_data[2].valid := 1, [1239].log_data[3].valid := 1, [1239].log_data[4].valid := 1, [1239].log_data[5].valid := 1, [1239].log_data[6].valid := 1, [1239].log_data[7].valid := 1, [1239].log_data[8].valid := 1, [1239].log_data[9].valid := 1, [1239].log_data[10].valid := 1, [1239].log_data[11].valid := 1, [1239].log_data[12].valid := 1, [1239].log_data[13].valid := 1, [1239].log_data[14].valid := 1, [1239].log_data[15].valid := 1, [1239].log_data[16].valid := 1, [1239].log_data[17].valid := 1, [1239].log_data[18].valid := 1, [1239].log_data[19].valid := 1, [1239].time.Year := 2023, [1239].time.Month := 1,
        [1239].time.Day := 13, [1239].time.Hour := 23, [1239].time.Minute := 39, [1239].time.Second := 59, [1240].log_data[0].min := 1.0, [1240].log_data[0].max := 1.0, [1240].log_data[0].total := 300.0, [1240].log_data[0].time := 300.0, [1240].log_data[0].minminute := 40, [1240].log_data[0].maxminute := 40, [1240].log_data[0].valid := 1, [1240].log_data[1].valid := 1, [1240].log_data[2].valid := 1, [1240].log_data[3].valid := 1, [1240].log_data[4].valid := 1, [1240].log_data[5].valid := 1, [1240].log_data[6].valid := 1, [1240].log_data[7].valid := 1, [1240].log_data[8].valid := 1, [1240].log_data[9].valid := 1, [1240].log_data[10].valid := 1, [1240].log_data[11].valid := 1, [1240].log_data[12].valid := 1, [1240].log_data[13].valid := 1, [1240].log_data[14].valid := 1, [1240].log_data[15].valid := 1, [1240].log_data[16].valid := 1, [1240].log_data[17].valid := 1, [1240].log_data[18].valid := 1, [1240].log_data[19].valid := 1, [1240].time.Year := 2023, [1240].time.Month := 1, [1240].time.Day := 13, [1240].time.Hour := 23, [1240].time.Minute := 44, [1240].time.Second := 59, [1241].log_data[0].min := 1.0, [1241].log_data[0].max := 1.0, [1241].log_data[0].total := 300.0, [1241].log_data[0].time := 300.0, [1241].log_data[0].minminute := 45, [1241].log_data[0].maxminute := 45, [1241].log_data[0].valid := 1, [1241].log_data[1].valid := 1, [1241].log_data[2].valid := 1, [1241].log_data[3].valid := 1, [1241].log_data[4].valid := 1, [1241].log_data[5].valid := 1, [1241].log_data[6].valid := 1, [1241].log_data[7].valid := 1, [1241].log_data[8].valid := 1, [1241].log_data[9].valid := 1, [1241].log_data[10].valid := 1, [1241].log_data[11].valid := 1, [1241].log_data[12].valid := 1, [1241].log_data[13].valid := 1, [1241].log_data[14].valid := 1, [1241].log_data[15].valid := 1, [1241].log_data[16].valid := 1, [1241].log_data[17].valid := 1,
        [1241].log_data[18].valid := 1, [1241].log_data[19].valid := 1, [1241].time.Year := 2023, [1241].time.Month := 1, [1241].time.Day := 13, [1241].time.Hour := 23, [1241].time.Minute := 49, [1241].time.Second := 59, [1242].log_data[0].min := 1.0, [1242].log_data[0].max := 1.0, [1242].log_data[0].total := 300.0, [1242].log_data[0].time := 300.0, [1242].log_data[0].minminute := 50, [1242].log_data[0].maxminute := 50, [1242].log_data[0].valid := 1, [1242].log_data[1].valid := 1, [1242].log_data[2].valid := 1, [1242].log_data[3].valid := 1, [1242].log_data[4].valid := 1, [1242].log_data[5].valid := 1, [1242].log_data[6].valid := 1, [1242].log_data[7].valid := 1, [1242].log_data[8].valid := 1, [1242].log_data[9].valid := 1, [1242].log_data[10].valid := 1, [1242].log_data[11].valid := 1, [1242].log_data[12].valid := 1, [1242].log_data[13].valid := 1, [1242].log_data[14].valid := 1, [1242].log_data[15].valid := 1, [1242].log_data[16].valid := 1, [1242].log_data[17].valid := 1, [1242].log_data[18].valid := 1, [1242].log_data[19].valid := 1, [1242].time.Year := 2023, [1242].time.Month := 1, [1242].time.Day := 13, [1242].time.Hour := 23, [1242].time.Minute := 54, [1242].time.Second := 59, [1243].log_data[0].min := 1.0, [1243].log_data[0].max := 1.0, [1243].log_data[0].total := 300.0, [1243].log_data[0].time := 300.0, [1243].log_data[0].minminute := 55, [1243].log_data[0].maxminute := 55, [1243].log_data[0].valid := 1, [1243].log_data[1].valid := 1, [1243].log_data[2].valid := 1, [1243].log_data[3].valid := 1, [1243].log_data[4].valid := 1, [1243].log_data[5].valid := 1, [1243].log_data[6].valid := 1, [1243].log_data[7].valid := 1, [1243].log_data[8].valid := 1, [1243].log_data[9].valid := 1, [1243].log_data[10].valid := 1, [1243].log_data[11].valid := 1, [1243].log_data[12].valid := 1, [1243].log_data[13].valid := 1,
        [1243].log_data[14].valid := 1, [1243].log_data[15].valid := 1, [1243].log_data[16].valid := 1, [1243].log_data[17].valid := 1, [1243].log_data[18].valid := 1, [1243].log_data[19].valid := 1, [1243].time.Year := 2023, [1243].time.Month := 1, [1243].time.Day := 13, [1243].time.Hour := 23, [1243].time.Minute := 59, [1243].time.Second := 59, [1244].log_data[0].min := 1.0, [1244].log_data[0].max := 1.0, [1244].log_data[0].total := 299.5, [1244].log_data[0].time := 299.5, [1244].log_data[0].valid := 1, [1244].log_data[1].valid := 1, [1244].log_data[2].valid := 1, [1244].log_data[3].valid := 1, [1244].log_data[4].valid := 1, [1244].log_data[5].valid := 1, [1244].log_data[6].valid := 1, [1244].log_data[7].valid := 1, [1244].log_data[8].valid := 1, [1244].log_data[9].valid := 1, [1244].log_data[10].valid := 1, [1244].log_data[11].valid := 1, [1244].log_data[12].valid := 1, [1244].log_data[13].valid := 1, [1244].log_data[14].valid := 1, [1244].log_data[15].valid := 1, [1244].log_data[16].valid := 1, [1244].log_data[17].valid := 1, [1244].log_data[18].valid := 1, [1244].log_data[19].valid := 1, [1244].time.Year := 2023, [1244].time.Month := 1, [1244].time.Day := 14, [1244].time.Minute := 4, [1244].time.Second := 59, [1245].log_data[0].min := 1.0, [1245].log_data[0].max := 1.0, [1245].log_data[0].total := 300.0, [1245].log_data[0].time := 300.0, [1245].log_data[0].minminute := 5, [1245].log_data[0].maxminute := 5, [1245].log_data[0].valid := 1, [1245].log_data[1].valid := 1, [1245].log_data[2].valid := 1, [1245].log_data[3].valid := 1, [1245].log_data[4].valid := 1, [1245].log_data[5].valid := 1, [1245].log_data[6].valid := 1, [1245].log_data[7].valid := 1, [1245].log_data[8].valid := 1, [1245].log_data[9].valid := 1, [1245].log_data[10].valid := 1, [1245].log_data[11].valid := 1, [1245].log_data[12].valid := 1,
        [1245].log_data[13].valid := 1, [1245].log_data[14].valid := 1, [1245].log_data[15].valid := 1, [1245].log_data[16].valid := 1, [1245].log_data[17].valid := 1, [1245].log_data[18].valid := 1, [1245].log_data[19].valid := 1, [1245].time.Year := 2023, [1245].time.Month := 1, [1245].time.Day := 14, [1245].time.Minute := 9, [1245].time.Second := 59, [1246].log_data[0].min := 1.0, [1246].log_data[0].max := 1.0, [1246].log_data[0].total := 300.0, [1246].log_data[0].time := 300.0, [1246].log_data[0].minminute := 10, [1246].log_data[0].maxminute := 10, [1246].log_data[0].valid := 1, [1246].log_data[1].valid := 1, [1246].log_data[2].valid := 1, [1246].log_data[3].valid := 1, [1246].log_data[4].valid := 1, [1246].log_data[5].valid := 1, [1246].log_data[6].valid := 1, [1246].log_data[7].valid := 1, [1246].log_data[8].valid := 1, [1246].log_data[9].valid := 1, [1246].log_data[10].valid := 1, [1246].log_data[11].valid := 1, [1246].log_data[12].valid := 1, [1246].log_data[13].valid := 1, [1246].log_data[14].valid := 1, [1246].log_data[15].valid := 1, [1246].log_data[16].valid := 1, [1246].log_data[17].valid := 1, [1246].log_data[18].valid := 1, [1246].log_data[19].valid := 1, [1246].time.Year := 2023, [1246].time.Month := 1, [1246].time.Day := 14, [1246].time.Minute := 14, [1246].time.Second := 59, [1247].log_data[0].min := 1.0, [1247].log_data[0].max := 1.0, [1247].log_data[0].total := 300.0, [1247].log_data[0].time := 300.0, [1247].log_data[0].minminute := 15, [1247].log_data[0].maxminute := 15, [1247].log_data[0].valid := 1, [1247].log_data[1].valid := 1, [1247].log_data[2].valid := 1, [1247].log_data[3].valid := 1, [1247].log_data[4].valid := 1, [1247].log_data[5].valid := 1, [1247].log_data[6].valid := 1, [1247].log_data[7].valid := 1, [1247].log_data[8].valid := 1, [1247].log_data[9].valid := 1, [1247].log_data[10].valid := 1,
        [1247].log_data[11].valid := 1, [1247].log_data[12].valid := 1, [1247].log_data[13].valid := 1, [1247].log_data[14].valid := 1, [1247].log_data[15].valid := 1, [1247].log_data[16].valid := 1, [1247].log_data[17].valid := 1, [1247].log_data[18].valid := 1, [1247].log_data[19].valid := 1, [1247].time.Year := 2023, [1247].time.Month := 1, [1247].time.Day := 14, [1247].time.Minute := 19, [1247].time.Second := 59, [1248].log_data[0].min := 1.0, [1248].log_data[0].max := 1.0, [1248].log_data[0].total := 300.0, [1248].log_data[0].time := 300.0, [1248].log_data[0].minminute := 20, [1248].log_data[0].maxminute := 20, [1248].log_data[0].valid := 1, [1248].log_data[1].valid := 1, [1248].log_data[2].valid := 1, [1248].log_data[3].valid := 1, [1248].log_data[4].valid := 1, [1248].log_data[5].valid := 1, [1248].log_data[6].valid := 1, [1248].log_data[7].valid := 1, [1248].log_data[8].valid := 1, [1248].log_data[9].valid := 1, [1248].log_data[10].valid := 1, [1248].log_data[11].valid := 1, [1248].log_data[12].valid := 1, [1248].log_data[13].valid := 1, [1248].log_data[14].valid := 1, [1248].log_data[15].valid := 1, [1248].log_data[16].valid := 1, [1248].log_data[17].valid := 1, [1248].log_data[18].valid := 1, [1248].log_data[19].valid := 1, [1248].time.Year := 2023, [1248].time.Month := 1, [1248].time.Day := 14, [1248].time.Minute := 24, [1248].time.Second := 59, [1249].log_data[0].min := 1.0, [1249].log_data[0].max := 1.0, [1249].log_data[0].total := 300.0, [1249].log_data[0].time := 300.0, [1249].log_data[0].minminute := 25, [1249].log_data[0].maxminute := 25, [1249].log_data[0].valid := 1, [1249].log_data[1].valid := 1, [1249].log_data[2].valid := 1, [1249].log_data[3].valid := 1, [1249].log_data[4].valid := 1, [1249].log_data[5].valid := 1, [1249].log_data[6].valid := 1, [1249].log_data[7].valid := 1, [1249].log_data[8].valid := 1,
        [1249].log_data[9].valid := 1, [1249].log_data[10].valid := 1, [1249].log_data[11].valid := 1, [1249].log_data[12].valid := 1, [1249].log_data[13].valid := 1, [1249].log_data[14].valid := 1, [1249].log_data[15].valid := 1, [1249].log_data[16].valid := 1, [1249].log_data[17].valid := 1, [1249].log_data[18].valid := 1, [1249].log_data[19].valid := 1, [1249].time.Year := 2023, [1249].time.Month := 1, [1249].time.Day := 14, [1249].time.Minute := 29, [1249].time.Second := 59, [1250].log_data[0].min := 1.0, [1250].log_data[0].max := 1.0, [1250].log_data[0].total := 300.0, [1250].log_data[0].time := 300.0, [1250].log_data[0].minminute := 30, [1250].log_data[0].maxminute := 30, [1250].log_data[0].valid := 1, [1250].log_data[1].valid := 1, [1250].log_data[2].valid := 1, [1250].log_data[3].valid := 1, [1250].log_data[4].valid := 1, [1250].log_data[5].valid := 1, [1250].log_data[6].valid := 1, [1250].log_data[7].valid := 1, [1250].log_data[8].valid := 1, [1250].log_data[9].valid := 1, [1250].log_data[10].valid := 1, [1250].log_data[11].valid := 1, [1250].log_data[12].valid := 1, [1250].log_data[13].valid := 1, [1250].log_data[14].valid := 1, [1250].log_data[15].valid := 1, [1250].log_data[16].valid := 1, [1250].log_data[17].valid := 1, [1250].log_data[18].valid := 1, [1250].log_data[19].valid := 1, [1250].time.Year := 2023, [1250].time.Month := 1, [1250].time.Day := 14, [1250].time.Minute := 34, [1250].time.Second := 59, [1251].log_data[0].min := 1.0, [1251].log_data[0].max := 1.0, [1251].log_data[0].total := 300.0, [1251].log_data[0].time := 300.0, [1251].log_data[0].minminute := 35, [1251].log_data[0].maxminute := 35, [1251].log_data[0].valid := 1, [1251].log_data[1].valid := 1, [1251].log_data[2].valid := 1, [1251].log_data[3].valid := 1, [1251].log_data[4].valid := 1, [1251].log_data[5].valid := 1, [1251].log_data[6].valid := 1,
        [1251].log_data[7].valid := 1, [1251].log_data[8].valid := 1, [1251].log_data[9].valid := 1, [1251].log_data[10].valid := 1, [1251].log_data[11].valid := 1, [1251].log_data[12].valid := 1, [1251].log_data[13].valid := 1, [1251].log_data[14].valid := 1, [1251].log_data[15].valid := 1, [1251].log_data[16].valid := 1, [1251].log_data[17].valid := 1, [1251].log_data[18].valid := 1, [1251].log_data[19].valid := 1, [1251].time.Year := 2023, [1251].time.Month := 1, [1251].time.Day := 14, [1251].time.Minute := 39, [1251].time.Second := 59, [1252].log_data[0].min := 1.0, [1252].log_data[0].max := 1.0, [1252].log_data[0].total := 300.0, [1252].log_data[0].time := 300.0, [1252].log_data[0].minminute := 40, [1252].log_data[0].maxminute := 40, [1252].log_data[0].valid := 1, [1252].log_data[1].valid := 1, [1252].log_data[2].valid := 1, [1252].log_data[3].valid := 1, [1252].log_data[4].valid := 1, [1252].log_data[5].valid := 1, [1252].log_data[6].valid := 1, [1252].log_data[7].valid := 1, [1252].log_data[8].valid := 1, [1252].log_data[9].valid := 1, [1252].log_data[10].valid := 1, [1252].log_data[11].valid := 1, [1252].log_data[12].valid := 1, [1252].log_data[13].valid := 1, [1252].log_data[14].valid := 1, [1252].log_data[15].valid := 1, [1252].log_data[16].valid := 1, [1252].log_data[17].valid := 1, [1252].log_data[18].valid := 1, [1252].log_data[19].valid := 1, [1252].time.Year := 2023, [1252].time.Month := 1, [1252].time.Day := 14, [1252].time.Minute := 44, [1252].time.Second := 59, [1253].log_data[0].min := 1.0, [1253].log_data[0].max := 1.0, [1253].log_data[0].total := 300.0, [1253].log_data[0].time := 300.0, [1253].log_data[0].minminute := 45, [1253].log_data[0].maxminute := 45, [1253].log_data[0].valid := 1, [1253].log_data[1].valid := 1, [1253].log_data[2].valid := 1, [1253].log_data[3].valid := 1, [1253].log_data[4].valid := 1,
        [1253].log_data[5].valid := 1, [1253].log_data[6].valid := 1, [1253].log_data[7].valid := 1, [1253].log_data[8].valid := 1, [1253].log_data[9].valid := 1, [1253].log_data[10].valid := 1, [1253].log_data[11].valid := 1, [1253].log_data[12].valid := 1, [1253].log_data[13].valid := 1, [1253].log_data[14].valid := 1, [1253].log_data[15].valid := 1, [1253].log_data[16].valid := 1, [1253].log_data[17].valid := 1, [1253].log_data[18].valid := 1, [1253].log_data[19].valid := 1, [1253].time.Year := 2023, [1253].time.Month := 1, [1253].time.Day := 14, [1253].time.Minute := 49, [1253].time.Second := 59, [1254].log_data[0].min := 1.0, [1254].log_data[0].max := 1.0, [1254].log_data[0].total := 300.0, [1254].log_data[0].time := 300.0, [1254].log_data[0].minminute := 50, [1254].log_data[0].maxminute := 50, [1254].log_data[0].valid := 1, [1254].log_data[1].valid := 1, [1254].log_data[2].valid := 1, [1254].log_data[3].valid := 1, [1254].log_data[4].valid := 1, [1254].log_data[5].valid := 1, [1254].log_data[6].valid := 1, [1254].log_data[7].valid := 1, [1254].log_data[8].valid := 1, [1254].log_data[9].valid := 1, [1254].log_data[10].valid := 1, [1254].log_data[11].valid := 1, [1254].log_data[12].valid := 1, [1254].log_data[13].valid := 1, [1254].log_data[14].valid := 1, [1254].log_data[15].valid := 1, [1254].log_data[16].valid := 1, [1254].log_data[17].valid := 1, [1254].log_data[18].valid := 1, [1254].log_data[19].valid := 1, [1254].time.Year := 2023, [1254].time.Month := 1, [1254].time.Day := 14, [1254].time.Minute := 54, [1254].time.Second := 59, [1255].log_data[0].min := 1.0, [1255].log_data[0].max := 1.0, [1255].log_data[0].total := 300.0, [1255].log_data[0].time := 300.0, [1255].log_data[0].minminute := 55, [1255].log_data[0].maxminute := 55, [1255].log_data[0].valid := 1, [1255].log_data[1].valid := 1, [1255].log_data[2].valid := 1,
        [1255].log_data[3].valid := 1, [1255].log_data[4].valid := 1, [1255].log_data[5].valid := 1, [1255].log_data[6].valid := 1, [1255].log_data[7].valid := 1, [1255].log_data[8].valid := 1, [1255].log_data[9].valid := 1, [1255].log_data[10].valid := 1, [1255].log_data[11].valid := 1, [1255].log_data[12].valid := 1, [1255].log_data[13].valid := 1, [1255].log_data[14].valid := 1, [1255].log_data[15].valid := 1, [1255].log_data[16].valid := 1, [1255].log_data[17].valid := 1, [1255].log_data[18].valid := 1, [1255].log_data[19].valid := 1, [1255].time.Year := 2023, [1255].time.Month := 1, [1255].time.Day := 14, [1255].time.Minute := 59, [1255].time.Second := 59, [1256].log_data[0].min := 1.0, [1256].log_data[0].max := 1.0, [1256].log_data[0].total := 300.0, [1256].log_data[0].time := 300.0, [1256].log_data[0].valid := 1, [1256].log_data[1].valid := 1, [1256].log_data[2].valid := 1, [1256].log_data[3].valid := 1, [1256].log_data[4].valid := 1, [1256].log_data[5].valid := 1, [1256].log_data[6].valid := 1, [1256].log_data[7].valid := 1, [1256].log_data[8].valid := 1, [1256].log_data[9].valid := 1, [1256].log_data[10].valid := 1, [1256].log_data[11].valid := 1, [1256].log_data[12].valid := 1, [1256].log_data[13].valid := 1, [1256].log_data[14].valid := 1, [1256].log_data[15].valid := 1, [1256].log_data[16].valid := 1, [1256].log_data[17].valid := 1, [1256].log_data[18].valid := 1, [1256].log_data[19].valid := 1, [1256].time.Year := 2023, [1256].time.Month := 1, [1256].time.Day := 14, [1256].time.Hour := 1, [1256].time.Minute := 4, [1256].time.Second := 59, [1257].log_data[0].min := 1.0, [1257].log_data[0].max := 1.0, [1257].log_data[0].total := 300.0, [1257].log_data[0].time := 300.0, [1257].log_data[0].minminute := 5, [1257].log_data[0].maxminute := 5, [1257].log_data[0].valid := 1, [1257].log_data[1].valid := 1,
        [1257].log_data[2].valid := 1, [1257].log_data[3].valid := 1, [1257].log_data[4].valid := 1, [1257].log_data[5].valid := 1, [1257].log_data[6].valid := 1, [1257].log_data[7].valid := 1, [1257].log_data[8].valid := 1, [1257].log_data[9].valid := 1, [1257].log_data[10].valid := 1, [1257].log_data[11].valid := 1, [1257].log_data[12].valid := 1, [1257].log_data[13].valid := 1, [1257].log_data[14].valid := 1, [1257].log_data[15].valid := 1, [1257].log_data[16].valid := 1, [1257].log_data[17].valid := 1, [1257].log_data[18].valid := 1, [1257].log_data[19].valid := 1, [1257].time.Year := 2023, [1257].time.Month := 1, [1257].time.Day := 14, [1257].time.Hour := 1, [1257].time.Minute := 9, [1257].time.Second := 59, [1258].log_data[0].min := 1.0, [1258].log_data[0].max := 1.0, [1258].log_data[0].total := 300.0, [1258].log_data[0].time := 300.0, [1258].log_data[0].minminute := 10, [1258].log_data[0].maxminute := 10, [1258].log_data[0].valid := 1, [1258].log_data[1].valid := 1, [1258].log_data[2].valid := 1, [1258].log_data[3].valid := 1, [1258].log_data[4].valid := 1, [1258].log_data[5].valid := 1, [1258].log_data[6].valid := 1, [1258].log_data[7].valid := 1, [1258].log_data[8].valid := 1, [1258].log_data[9].valid := 1, [1258].log_data[10].valid := 1, [1258].log_data[11].valid := 1, [1258].log_data[12].valid := 1, [1258].log_data[13].valid := 1, [1258].log_data[14].valid := 1, [1258].log_data[15].valid := 1, [1258].log_data[16].valid := 1, [1258].log_data[17].valid := 1, [1258].log_data[18].valid := 1, [1258].log_data[19].valid := 1, [1258].time.Year := 2023, [1258].time.Month := 1, [1258].time.Day := 14, [1258].time.Hour := 1, [1258].time.Minute := 14, [1258].time.Second := 59, [1259].log_data[0].min := 1.0, [1259].log_data[0].max := 1.0, [1259].log_data[0].total := 300.0, [1259].log_data[0].time := 300.0,
        [1259].log_data[0].minminute := 15, [1259].log_data[0].maxminute := 15, [1259].log_data[0].valid := 1, [1259].log_data[1].valid := 1, [1259].log_data[2].valid := 1, [1259].log_data[3].valid := 1, [1259].log_data[4].valid := 1, [1259].log_data[5].valid := 1, [1259].log_data[6].valid := 1, [1259].log_data[7].valid := 1, [1259].log_data[8].valid := 1, [1259].log_data[9].valid := 1, [1259].log_data[10].valid := 1, [1259].log_data[11].valid := 1, [1259].log_data[12].valid := 1, [1259].log_data[13].valid := 1, [1259].log_data[14].valid := 1, [1259].log_data[15].valid := 1, [1259].log_data[16].valid := 1, [1259].log_data[17].valid := 1, [1259].log_data[18].valid := 1, [1259].log_data[19].valid := 1, [1259].time.Year := 2023, [1259].time.Month := 1, [1259].time.Day := 14, [1259].time.Hour := 1, [1259].time.Minute := 19, [1259].time.Second := 59, [1260].log_data[0].min := 1.0, [1260].log_data[0].max := 1.0, [1260].log_data[0].total := 300.0, [1260].log_data[0].time := 300.0, [1260].log_data[0].minminute := 20, [1260].log_data[0].maxminute := 20, [1260].log_data[0].valid := 1, [1260].log_data[1].valid := 1, [1260].log_data[2].valid := 1, [1260].log_data[3].valid := 1, [1260].log_data[4].valid := 1, [1260].log_data[5].valid := 1, [1260].log_data[6].valid := 1, [1260].log_data[7].valid := 1, [1260].log_data[8].valid := 1, [1260].log_data[9].valid := 1, [1260].log_data[10].valid := 1, [1260].log_data[11].valid := 1, [1260].log_data[12].valid := 1, [1260].log_data[13].valid := 1, [1260].log_data[14].valid := 1, [1260].log_data[15].valid := 1, [1260].log_data[16].valid := 1, [1260].log_data[17].valid := 1, [1260].log_data[18].valid := 1, [1260].log_data[19].valid := 1, [1260].time.Year := 2023, [1260].time.Month := 1, [1260].time.Day := 14, [1260].time.Hour := 1, [1260].time.Minute := 24, [1260].time.Second := 59,
        [1261].log_data[0].min := 1.0, [1261].log_data[0].max := 1.0, [1261].log_data[0].total := 300.0, [1261].log_data[0].time := 300.0, [1261].log_data[0].minminute := 25, [1261].log_data[0].maxminute := 25, [1261].log_data[0].valid := 1, [1261].log_data[1].valid := 1, [1261].log_data[2].valid := 1, [1261].log_data[3].valid := 1, [1261].log_data[4].valid := 1, [1261].log_data[5].valid := 1, [1261].log_data[6].valid := 1, [1261].log_data[7].valid := 1, [1261].log_data[8].valid := 1, [1261].log_data[9].valid := 1, [1261].log_data[10].valid := 1, [1261].log_data[11].valid := 1, [1261].log_data[12].valid := 1, [1261].log_data[13].valid := 1, [1261].log_data[14].valid := 1, [1261].log_data[15].valid := 1, [1261].log_data[16].valid := 1, [1261].log_data[17].valid := 1, [1261].log_data[18].valid := 1, [1261].log_data[19].valid := 1, [1261].time.Year := 2023, [1261].time.Month := 1, [1261].time.Day := 14, [1261].time.Hour := 1, [1261].time.Minute := 29, [1261].time.Second := 59, [1262].log_data[0].min := 1.0, [1262].log_data[0].max := 1.0, [1262].log_data[0].total := 300.0, [1262].log_data[0].time := 300.0, [1262].log_data[0].minminute := 30, [1262].log_data[0].maxminute := 30, [1262].log_data[0].valid := 1, [1262].log_data[1].valid := 1, [1262].log_data[2].valid := 1, [1262].log_data[3].valid := 1, [1262].log_data[4].valid := 1, [1262].log_data[5].valid := 1, [1262].log_data[6].valid := 1, [1262].log_data[7].valid := 1, [1262].log_data[8].valid := 1, [1262].log_data[9].valid := 1, [1262].log_data[10].valid := 1, [1262].log_data[11].valid := 1, [1262].log_data[12].valid := 1, [1262].log_data[13].valid := 1, [1262].log_data[14].valid := 1, [1262].log_data[15].valid := 1, [1262].log_data[16].valid := 1, [1262].log_data[17].valid := 1, [1262].log_data[18].valid := 1, [1262].log_data[19].valid := 1, [1262].time.Year := 2023, [1262].time.Month := 1,
        [1262].time.Day := 14, [1262].time.Hour := 1, [1262].time.Minute := 34, [1262].time.Second := 59, [1263].log_data[0].min := 1.0, [1263].log_data[0].max := 1.0, [1263].log_data[0].total := 300.0, [1263].log_data[0].time := 300.0, [1263].log_data[0].minminute := 35, [1263].log_data[0].maxminute := 35, [1263].log_data[0].valid := 1, [1263].log_data[1].valid := 1, [1263].log_data[2].valid := 1, [1263].log_data[3].valid := 1, [1263].log_data[4].valid := 1, [1263].log_data[5].valid := 1, [1263].log_data[6].valid := 1, [1263].log_data[7].valid := 1, [1263].log_data[8].valid := 1, [1263].log_data[9].valid := 1, [1263].log_data[10].valid := 1, [1263].log_data[11].valid := 1, [1263].log_data[12].valid := 1, [1263].log_data[13].valid := 1, [1263].log_data[14].valid := 1, [1263].log_data[15].valid := 1, [1263].log_data[16].valid := 1, [1263].log_data[17].valid := 1, [1263].log_data[18].valid := 1, [1263].log_data[19].valid := 1, [1263].time.Year := 2023, [1263].time.Month := 1, [1263].time.Day := 14, [1263].time.Hour := 1, [1263].time.Minute := 39, [1263].time.Second := 59, [1264].log_data[0].min := 1.0, [1264].log_data[0].max := 1.0, [1264].log_data[0].total := 300.0, [1264].log_data[0].time := 300.0, [1264].log_data[0].minminute := 40, [1264].log_data[0].maxminute := 40, [1264].log_data[0].valid := 1, [1264].log_data[1].valid := 1, [1264].log_data[2].valid := 1, [1264].log_data[3].valid := 1, [1264].log_data[4].valid := 1, [1264].log_data[5].valid := 1, [1264].log_data[6].valid := 1, [1264].log_data[7].valid := 1, [1264].log_data[8].valid := 1, [1264].log_data[9].valid := 1, [1264].log_data[10].valid := 1, [1264].log_data[11].valid := 1, [1264].log_data[12].valid := 1, [1264].log_data[13].valid := 1, [1264].log_data[14].valid := 1, [1264].log_data[15].valid := 1, [1264].log_data[16].valid := 1, [1264].log_data[17].valid := 1,
        [1264].log_data[18].valid := 1, [1264].log_data[19].valid := 1, [1264].time.Year := 2023, [1264].time.Month := 1, [1264].time.Day := 14, [1264].time.Hour := 1, [1264].time.Minute := 44, [1264].time.Second := 59, [1265].log_data[0].min := 1.0, [1265].log_data[0].max := 1.0, [1265].log_data[0].total := 300.0, [1265].log_data[0].time := 300.0, [1265].log_data[0].minminute := 45, [1265].log_data[0].maxminute := 45, [1265].log_data[0].valid := 1, [1265].log_data[1].valid := 1, [1265].log_data[2].valid := 1, [1265].log_data[3].valid := 1, [1265].log_data[4].valid := 1, [1265].log_data[5].valid := 1, [1265].log_data[6].valid := 1, [1265].log_data[7].valid := 1, [1265].log_data[8].valid := 1, [1265].log_data[9].valid := 1, [1265].log_data[10].valid := 1, [1265].log_data[11].valid := 1, [1265].log_data[12].valid := 1, [1265].log_data[13].valid := 1, [1265].log_data[14].valid := 1, [1265].log_data[15].valid := 1, [1265].log_data[16].valid := 1, [1265].log_data[17].valid := 1, [1265].log_data[18].valid := 1, [1265].log_data[19].valid := 1, [1265].time.Year := 2023, [1265].time.Month := 1, [1265].time.Day := 14, [1265].time.Hour := 1, [1265].time.Minute := 49, [1265].time.Second := 59, [1266].log_data[0].min := 1.0, [1266].log_data[0].max := 1.0, [1266].log_data[0].total := 300.0, [1266].log_data[0].time := 300.0, [1266].log_data[0].minminute := 50, [1266].log_data[0].maxminute := 50, [1266].log_data[0].valid := 1, [1266].log_data[1].valid := 1, [1266].log_data[2].valid := 1, [1266].log_data[3].valid := 1, [1266].log_data[4].valid := 1, [1266].log_data[5].valid := 1, [1266].log_data[6].valid := 1, [1266].log_data[7].valid := 1, [1266].log_data[8].valid := 1, [1266].log_data[9].valid := 1, [1266].log_data[10].valid := 1, [1266].log_data[11].valid := 1, [1266].log_data[12].valid := 1, [1266].log_data[13].valid := 1,
        [1266].log_data[14].valid := 1, [1266].log_data[15].valid := 1, [1266].log_data[16].valid := 1, [1266].log_data[17].valid := 1, [1266].log_data[18].valid := 1, [1266].log_data[19].valid := 1, [1266].time.Year := 2023, [1266].time.Month := 1, [1266].time.Day := 14, [1266].time.Hour := 1, [1266].time.Minute := 54, [1266].time.Second := 59, [1267].log_data[0].min := 1.0, [1267].log_data[0].max := 1.0, [1267].log_data[0].total := 300.0, [1267].log_data[0].time := 300.0, [1267].log_data[0].minminute := 55, [1267].log_data[0].maxminute := 55, [1267].log_data[0].valid := 1, [1267].log_data[1].valid := 1, [1267].log_data[2].valid := 1, [1267].log_data[3].valid := 1, [1267].log_data[4].valid := 1, [1267].log_data[5].valid := 1, [1267].log_data[6].valid := 1, [1267].log_data[7].valid := 1, [1267].log_data[8].valid := 1, [1267].log_data[9].valid := 1, [1267].log_data[10].valid := 1, [1267].log_data[11].valid := 1, [1267].log_data[12].valid := 1, [1267].log_data[13].valid := 1, [1267].log_data[14].valid := 1, [1267].log_data[15].valid := 1, [1267].log_data[16].valid := 1, [1267].log_data[17].valid := 1, [1267].log_data[18].valid := 1, [1267].log_data[19].valid := 1, [1267].time.Year := 2023, [1267].time.Month := 1, [1267].time.Day := 14, [1267].time.Hour := 1, [1267].time.Minute := 59, [1267].time.Second := 59, [1268].log_data[0].min := 1.0, [1268].log_data[0].max := 1.0, [1268].log_data[0].total := 300.0, [1268].log_data[0].time := 300.0, [1268].log_data[0].valid := 1, [1268].log_data[1].valid := 1, [1268].log_data[2].valid := 1, [1268].log_data[3].valid := 1, [1268].log_data[4].valid := 1, [1268].log_data[5].valid := 1, [1268].log_data[6].valid := 1, [1268].log_data[7].valid := 1, [1268].log_data[8].valid := 1, [1268].log_data[9].valid := 1, [1268].log_data[10].valid := 1, [1268].log_data[11].valid := 1,
        [1268].log_data[12].valid := 1, [1268].log_data[13].valid := 1, [1268].log_data[14].valid := 1, [1268].log_data[15].valid := 1, [1268].log_data[16].valid := 1, [1268].log_data[17].valid := 1, [1268].log_data[18].valid := 1, [1268].log_data[19].valid := 1, [1268].time.Year := 2023, [1268].time.Month := 1, [1268].time.Day := 14, [1268].time.Hour := 2, [1268].time.Minute := 4, [1268].time.Second := 59, [1269].log_data[0].min := 1.0, [1269].log_data[0].max := 1.0, [1269].log_data[0].total := 300.0, [1269].log_data[0].time := 300.0, [1269].log_data[0].minminute := 5, [1269].log_data[0].maxminute := 5, [1269].log_data[0].valid := 1, [1269].log_data[1].valid := 1, [1269].log_data[2].valid := 1, [1269].log_data[3].valid := 1, [1269].log_data[4].valid := 1, [1269].log_data[5].valid := 1, [1269].log_data[6].valid := 1, [1269].log_data[7].valid := 1, [1269].log_data[8].valid := 1, [1269].log_data[9].valid := 1, [1269].log_data[10].valid := 1, [1269].log_data[11].valid := 1, [1269].log_data[12].valid := 1, [1269].log_data[13].valid := 1, [1269].log_data[14].valid := 1, [1269].log_data[15].valid := 1, [1269].log_data[16].valid := 1, [1269].log_data[17].valid := 1, [1269].log_data[18].valid := 1, [1269].log_data[19].valid := 1, [1269].time.Year := 2023, [1269].time.Month := 1, [1269].time.Day := 14, [1269].time.Hour := 2, [1269].time.Minute := 9, [1269].time.Second := 59, [1270].log_data[0].min := 1.0, [1270].log_data[0].max := 1.0, [1270].log_data[0].total := 300.0, [1270].log_data[0].time := 300.0, [1270].log_data[0].minminute := 10, [1270].log_data[0].maxminute := 10, [1270].log_data[0].valid := 1, [1270].log_data[1].valid := 1, [1270].log_data[2].valid := 1, [1270].log_data[3].valid := 1, [1270].log_data[4].valid := 1, [1270].log_data[5].valid := 1, [1270].log_data[6].valid := 1, [1270].log_data[7].valid := 1,
        [1270].log_data[8].valid := 1, [1270].log_data[9].valid := 1, [1270].log_data[10].valid := 1, [1270].log_data[11].valid := 1, [1270].log_data[12].valid := 1, [1270].log_data[13].valid := 1, [1270].log_data[14].valid := 1, [1270].log_data[15].valid := 1, [1270].log_data[16].valid := 1, [1270].log_data[17].valid := 1, [1270].log_data[18].valid := 1, [1270].log_data[19].valid := 1, [1270].time.Year := 2023, [1270].time.Month := 1, [1270].time.Day := 14, [1270].time.Hour := 2, [1270].time.Minute := 14, [1270].time.Second := 59, [1271].log_data[0].min := 1.0, [1271].log_data[0].max := 1.0, [1271].log_data[0].total := 300.0, [1271].log_data[0].time := 300.0, [1271].log_data[0].minminute := 15, [1271].log_data[0].maxminute := 15, [1271].log_data[0].valid := 1, [1271].log_data[1].valid := 1, [1271].log_data[2].valid := 1, [1271].log_data[3].valid := 1, [1271].log_data[4].valid := 1, [1271].log_data[5].valid := 1, [1271].log_data[6].valid := 1, [1271].log_data[7].valid := 1, [1271].log_data[8].valid := 1, [1271].log_data[9].valid := 1, [1271].log_data[10].valid := 1, [1271].log_data[11].valid := 1, [1271].log_data[12].valid := 1, [1271].log_data[13].valid := 1, [1271].log_data[14].valid := 1, [1271].log_data[15].valid := 1, [1271].log_data[16].valid := 1, [1271].log_data[17].valid := 1, [1271].log_data[18].valid := 1, [1271].log_data[19].valid := 1, [1271].time.Year := 2023, [1271].time.Month := 1, [1271].time.Day := 14, [1271].time.Hour := 2, [1271].time.Minute := 19, [1271].time.Second := 59, [1272].log_data[0].min := 1.0, [1272].log_data[0].max := 1.0, [1272].log_data[0].total := 300.0, [1272].log_data[0].time := 300.0, [1272].log_data[0].minminute := 20, [1272].log_data[0].maxminute := 20, [1272].log_data[0].valid := 1, [1272].log_data[1].valid := 1, [1272].log_data[2].valid := 1, [1272].log_data[3].valid := 1,
        [1272].log_data[4].valid := 1, [1272].log_data[5].valid := 1, [1272].log_data[6].valid := 1, [1272].log_data[7].valid := 1, [1272].log_data[8].valid := 1, [1272].log_data[9].valid := 1, [1272].log_data[10].valid := 1, [1272].log_data[11].valid := 1, [1272].log_data[12].valid := 1, [1272].log_data[13].valid := 1, [1272].log_data[14].valid := 1, [1272].log_data[15].valid := 1, [1272].log_data[16].valid := 1, [1272].log_data[17].valid := 1, [1272].log_data[18].valid := 1, [1272].log_data[19].valid := 1, [1272].time.Year := 2023, [1272].time.Month := 1, [1272].time.Day := 14, [1272].time.Hour := 2, [1272].time.Minute := 24, [1272].time.Second := 59, [1273].log_data[0].min := 1.0, [1273].log_data[0].max := 1.0, [1273].log_data[0].total := 300.0, [1273].log_data[0].time := 300.0, [1273].log_data[0].minminute := 25, [1273].log_data[0].maxminute := 25, [1273].log_data[0].valid := 1, [1273].log_data[1].valid := 1, [1273].log_data[2].valid := 1, [1273].log_data[3].valid := 1, [1273].log_data[4].valid := 1, [1273].log_data[5].valid := 1, [1273].log_data[6].valid := 1, [1273].log_data[7].valid := 1, [1273].log_data[8].valid := 1, [1273].log_data[9].valid := 1, [1273].log_data[10].valid := 1, [1273].log_data[11].valid := 1, [1273].log_data[12].valid := 1, [1273].log_data[13].valid := 1, [1273].log_data[14].valid := 1, [1273].log_data[15].valid := 1, [1273].log_data[16].valid := 1, [1273].log_data[17].valid := 1, [1273].log_data[18].valid := 1, [1273].log_data[19].valid := 1, [1273].time.Year := 2023, [1273].time.Month := 1, [1273].time.Day := 14, [1273].time.Hour := 2, [1273].time.Minute := 29, [1273].time.Second := 59, [1274].log_data[0].min := 1.0, [1274].log_data[0].max := 1.0, [1274].log_data[0].total := 300.0, [1274].log_data[0].time := 300.0, [1274].log_data[0].minminute := 30, [1274].log_data[0].maxminute := 30,
        [1274].log_data[0].valid := 1, [1274].log_data[1].valid := 1, [1274].log_data[2].valid := 1, [1274].log_data[3].valid := 1, [1274].log_data[4].valid := 1, [1274].log_data[5].valid := 1, [1274].log_data[6].valid := 1, [1274].log_data[7].valid := 1, [1274].log_data[8].valid := 1, [1274].log_data[9].valid := 1, [1274].log_data[10].valid := 1, [1274].log_data[11].valid := 1, [1274].log_data[12].valid := 1, [1274].log_data[13].valid := 1, [1274].log_data[14].valid := 1, [1274].log_data[15].valid := 1, [1274].log_data[16].valid := 1, [1274].log_data[17].valid := 1, [1274].log_data[18].valid := 1, [1274].log_data[19].valid := 1, [1274].time.Year := 2023, [1274].time.Month := 1, [1274].time.Day := 14, [1274].time.Hour := 2, [1274].time.Minute := 34, [1274].time.Second := 59, [1275].log_data[0].min := 1.0, [1275].log_data[0].max := 1.0, [1275].log_data[0].total := 300.0, [1275].log_data[0].time := 300.0, [1275].log_data[0].minminute := 35, [1275].log_data[0].maxminute := 35, [1275].log_data[0].valid := 1, [1275].log_data[1].valid := 1, [1275].log_data[2].valid := 1, [1275].log_data[3].valid := 1, [1275].log_data[4].valid := 1, [1275].log_data[5].valid := 1, [1275].log_data[6].valid := 1, [1275].log_data[7].valid := 1, [1275].log_data[8].valid := 1, [1275].log_data[9].valid := 1, [1275].log_data[10].valid := 1, [1275].log_data[11].valid := 1, [1275].log_data[12].valid := 1, [1275].log_data[13].valid := 1, [1275].log_data[14].valid := 1, [1275].log_data[15].valid := 1, [1275].log_data[16].valid := 1, [1275].log_data[17].valid := 1, [1275].log_data[18].valid := 1, [1275].log_data[19].valid := 1, [1275].time.Year := 2023, [1275].time.Month := 1, [1275].time.Day := 14, [1275].time.Hour := 2, [1275].time.Minute := 39, [1275].time.Second := 59, [1276].log_data[0].min := 1.0, [1276].log_data[0].max := 1.0,
        [1276].log_data[0].total := 300.0, [1276].log_data[0].time := 300.0, [1276].log_data[0].minminute := 40, [1276].log_data[0].maxminute := 40, [1276].log_data[0].valid := 1, [1276].log_data[1].valid := 1, [1276].log_data[2].valid := 1, [1276].log_data[3].valid := 1, [1276].log_data[4].valid := 1, [1276].log_data[5].valid := 1, [1276].log_data[6].valid := 1, [1276].log_data[7].valid := 1, [1276].log_data[8].valid := 1, [1276].log_data[9].valid := 1, [1276].log_data[10].valid := 1, [1276].log_data[11].valid := 1, [1276].log_data[12].valid := 1, [1276].log_data[13].valid := 1, [1276].log_data[14].valid := 1, [1276].log_data[15].valid := 1, [1276].log_data[16].valid := 1, [1276].log_data[17].valid := 1, [1276].log_data[18].valid := 1, [1276].log_data[19].valid := 1, [1276].time.Year := 2023, [1276].time.Month := 1, [1276].time.Day := 14, [1276].time.Hour := 2, [1276].time.Minute := 44, [1276].time.Second := 59, [1277].log_data[0].min := 1.0, [1277].log_data[0].max := 1.0, [1277].log_data[0].total := 300.0, [1277].log_data[0].time := 300.0, [1277].log_data[0].minminute := 45, [1277].log_data[0].maxminute := 45, [1277].log_data[0].valid := 1, [1277].log_data[1].valid := 1, [1277].log_data[2].valid := 1, [1277].log_data[3].valid := 1, [1277].log_data[4].valid := 1, [1277].log_data[5].valid := 1, [1277].log_data[6].valid := 1, [1277].log_data[7].valid := 1, [1277].log_data[8].valid := 1, [1277].log_data[9].valid := 1, [1277].log_data[10].valid := 1, [1277].log_data[11].valid := 1, [1277].log_data[12].valid := 1, [1277].log_data[13].valid := 1, [1277].log_data[14].valid := 1, [1277].log_data[15].valid := 1, [1277].log_data[16].valid := 1, [1277].log_data[17].valid := 1, [1277].log_data[18].valid := 1, [1277].log_data[19].valid := 1, [1277].time.Year := 2023, [1277].time.Month := 1, [1277].time.Day := 14, [1277].time.Hour := 2,
        [1277].time.Minute := 49, [1277].time.Second := 59, [1278].log_data[0].min := 1.0, [1278].log_data[0].max := 1.0, [1278].log_data[0].total := 300.0, [1278].log_data[0].time := 300.0, [1278].log_data[0].minminute := 50, [1278].log_data[0].maxminute := 50, [1278].log_data[0].valid := 1, [1278].log_data[1].valid := 1, [1278].log_data[2].valid := 1, [1278].log_data[3].valid := 1, [1278].log_data[4].valid := 1, [1278].log_data[5].valid := 1, [1278].log_data[6].valid := 1, [1278].log_data[7].valid := 1, [1278].log_data[8].valid := 1, [1278].log_data[9].valid := 1, [1278].log_data[10].valid := 1, [1278].log_data[11].valid := 1, [1278].log_data[12].valid := 1, [1278].log_data[13].valid := 1, [1278].log_data[14].valid := 1, [1278].log_data[15].valid := 1, [1278].log_data[16].valid := 1, [1278].log_data[17].valid := 1, [1278].log_data[18].valid := 1, [1278].log_data[19].valid := 1, [1278].time.Year := 2023, [1278].time.Month := 1, [1278].time.Day := 14, [1278].time.Hour := 2, [1278].time.Minute := 54, [1278].time.Second := 59, [1279].log_data[0].min := 1.0, [1279].log_data[0].max := 1.0, [1279].log_data[0].total := 300.0, [1279].log_data[0].time := 300.0, [1279].log_data[0].minminute := 55, [1279].log_data[0].maxminute := 55, [1279].log_data[0].valid := 1, [1279].log_data[1].valid := 1, [1279].log_data[2].valid := 1, [1279].log_data[3].valid := 1, [1279].log_data[4].valid := 1, [1279].log_data[5].valid := 1, [1279].log_data[6].valid := 1, [1279].log_data[7].valid := 1, [1279].log_data[8].valid := 1, [1279].log_data[9].valid := 1, [1279].log_data[10].valid := 1, [1279].log_data[11].valid := 1, [1279].log_data[12].valid := 1, [1279].log_data[13].valid := 1, [1279].log_data[14].valid := 1, [1279].log_data[15].valid := 1, [1279].log_data[16].valid := 1, [1279].log_data[17].valid := 1, [1279].log_data[18].valid := 1, [1279].log_data[19].valid := 1,
        [1279].time.Year := 2023, [1279].time.Month := 1, [1279].time.Day := 14, [1279].time.Hour := 2, [1279].time.Minute := 59, [1279].time.Second := 59, [1280].log_data[0].min := 1.0, [1280].log_data[0].max := 1.0, [1280].log_data[0].total := 300.0, [1280].log_data[0].time := 300.0, [1280].log_data[0].valid := 1, [1280].log_data[1].valid := 1, [1280].log_data[2].valid := 1, [1280].log_data[3].valid := 1, [1280].log_data[4].valid := 1, [1280].log_data[5].valid := 1, [1280].log_data[6].valid := 1, [1280].log_data[7].valid := 1, [1280].log_data[8].valid := 1, [1280].log_data[9].valid := 1, [1280].log_data[10].valid := 1, [1280].log_data[11].valid := 1, [1280].log_data[12].valid := 1, [1280].log_data[13].valid := 1, [1280].log_data[14].valid := 1, [1280].log_data[15].valid := 1, [1280].log_data[16].valid := 1, [1280].log_data[17].valid := 1, [1280].log_data[18].valid := 1, [1280].log_data[19].valid := 1, [1280].time.Year := 2023, [1280].time.Month := 1, [1280].time.Day := 14, [1280].time.Hour := 3, [1280].time.Minute := 4, [1280].time.Second := 59, [1281].log_data[0].min := 1.0, [1281].log_data[0].max := 1.0, [1281].log_data[0].total := 300.0, [1281].log_data[0].time := 300.0, [1281].log_data[0].minminute := 5, [1281].log_data[0].maxminute := 5, [1281].log_data[0].valid := 1, [1281].log_data[1].valid := 1, [1281].log_data[2].valid := 1, [1281].log_data[3].valid := 1, [1281].log_data[4].valid := 1, [1281].log_data[5].valid := 1, [1281].log_data[6].valid := 1, [1281].log_data[7].valid := 1, [1281].log_data[8].valid := 1, [1281].log_data[9].valid := 1, [1281].log_data[10].valid := 1, [1281].log_data[11].valid := 1, [1281].log_data[12].valid := 1, [1281].log_data[13].valid := 1, [1281].log_data[14].valid := 1, [1281].log_data[15].valid := 1, [1281].log_data[16].valid := 1, [1281].log_data[17].valid := 1,
        [1281].log_data[18].valid := 1, [1281].log_data[19].valid := 1, [1281].time.Year := 2023, [1281].time.Month := 1, [1281].time.Day := 14, [1281].time.Hour := 3, [1281].time.Minute := 9, [1281].time.Second := 59, [1282].log_data[0].min := 1.0, [1282].log_data[0].max := 1.0, [1282].log_data[0].total := 300.0, [1282].log_data[0].time := 300.0, [1282].log_data[0].minminute := 10, [1282].log_data[0].maxminute := 10, [1282].log_data[0].valid := 1, [1282].log_data[1].valid := 1, [1282].log_data[2].valid := 1, [1282].log_data[3].valid := 1, [1282].log_data[4].valid := 1, [1282].log_data[5].valid := 1, [1282].log_data[6].valid := 1, [1282].log_data[7].valid := 1, [1282].log_data[8].valid := 1, [1282].log_data[9].valid := 1, [1282].log_data[10].valid := 1, [1282].log_data[11].valid := 1, [1282].log_data[12].valid := 1, [1282].log_data[13].valid := 1, [1282].log_data[14].valid := 1, [1282].log_data[15].valid := 1, [1282].log_data[16].valid := 1, [1282].log_data[17].valid := 1, [1282].log_data[18].valid := 1, [1282].log_data[19].valid := 1, [1282].time.Year := 2023, [1282].time.Month := 1, [1282].time.Day := 14, [1282].time.Hour := 3, [1282].time.Minute := 14, [1282].time.Second := 59, [1283].log_data[0].min := 1.0, [1283].log_data[0].max := 1.0, [1283].log_data[0].total := 300.0, [1283].log_data[0].time := 300.0, [1283].log_data[0].minminute := 15, [1283].log_data[0].maxminute := 15, [1283].log_data[0].valid := 1, [1283].log_data[1].valid := 1, [1283].log_data[2].valid := 1, [1283].log_data[3].valid := 1, [1283].log_data[4].valid := 1, [1283].log_data[5].valid := 1, [1283].log_data[6].valid := 1, [1283].log_data[7].valid := 1, [1283].log_data[8].valid := 1, [1283].log_data[9].valid := 1, [1283].log_data[10].valid := 1, [1283].log_data[11].valid := 1, [1283].log_data[12].valid := 1, [1283].log_data[13].valid := 1,
        [1283].log_data[14].valid := 1, [1283].log_data[15].valid := 1, [1283].log_data[16].valid := 1, [1283].log_data[17].valid := 1, [1283].log_data[18].valid := 1, [1283].log_data[19].valid := 1, [1283].time.Year := 2023, [1283].time.Month := 1, [1283].time.Day := 14, [1283].time.Hour := 3, [1283].time.Minute := 19, [1283].time.Second := 59, [1284].log_data[0].min := 1.0, [1284].log_data[0].max := 1.0, [1284].log_data[0].total := 300.0, [1284].log_data[0].time := 300.0, [1284].log_data[0].minminute := 20, [1284].log_data[0].maxminute := 20, [1284].log_data[0].valid := 1, [1284].log_data[1].valid := 1, [1284].log_data[2].valid := 1, [1284].log_data[3].valid := 1, [1284].log_data[4].valid := 1, [1284].log_data[5].valid := 1, [1284].log_data[6].valid := 1, [1284].log_data[7].valid := 1, [1284].log_data[8].valid := 1, [1284].log_data[9].valid := 1, [1284].log_data[10].valid := 1, [1284].log_data[11].valid := 1, [1284].log_data[12].valid := 1, [1284].log_data[13].valid := 1, [1284].log_data[14].valid := 1, [1284].log_data[15].valid := 1, [1284].log_data[16].valid := 1, [1284].log_data[17].valid := 1, [1284].log_data[18].valid := 1, [1284].log_data[19].valid := 1, [1284].time.Year := 2023, [1284].time.Month := 1, [1284].time.Day := 14, [1284].time.Hour := 3, [1284].time.Minute := 24, [1284].time.Second := 59, [1285].log_data[0].min := 1.0, [1285].log_data[0].max := 1.0, [1285].log_data[0].total := 300.0, [1285].log_data[0].time := 300.0, [1285].log_data[0].minminute := 25, [1285].log_data[0].maxminute := 25, [1285].log_data[0].valid := 1, [1285].log_data[1].valid := 1, [1285].log_data[2].valid := 1, [1285].log_data[3].valid := 1, [1285].log_data[4].valid := 1, [1285].log_data[5].valid := 1, [1285].log_data[6].valid := 1, [1285].log_data[7].valid := 1, [1285].log_data[8].valid := 1, [1285].log_data[9].valid := 1,
        [1285].log_data[10].valid := 1, [1285].log_data[11].valid := 1, [1285].log_data[12].valid := 1, [1285].log_data[13].valid := 1, [1285].log_data[14].valid := 1, [1285].log_data[15].valid := 1, [1285].log_data[16].valid := 1, [1285].log_data[17].valid := 1, [1285].log_data[18].valid := 1, [1285].log_data[19].valid := 1, [1285].time.Year := 2023, [1285].time.Month := 1, [1285].time.Day := 14, [1285].time.Hour := 3, [1285].time.Minute := 29, [1285].time.Second := 59, [1286].log_data[0].min := 1.0, [1286].log_data[0].max := 1.0, [1286].log_data[0].total := 300.0, [1286].log_data[0].time := 300.0, [1286].log_data[0].minminute := 30, [1286].log_data[0].maxminute := 30, [1286].log_data[0].valid := 1, [1286].log_data[1].valid := 1, [1286].log_data[2].valid := 1, [1286].log_data[3].valid := 1, [1286].log_data[4].valid := 1, [1286].log_data[5].valid := 1, [1286].log_data[6].valid := 1, [1286].log_data[7].valid := 1, [1286].log_data[8].valid := 1, [1286].log_data[9].valid := 1, [1286].log_data[10].valid := 1, [1286].log_data[11].valid := 1, [1286].log_data[12].valid := 1, [1286].log_data[13].valid := 1, [1286].log_data[14].valid := 1, [1286].log_data[15].valid := 1, [1286].log_data[16].valid := 1, [1286].log_data[17].valid := 1, [1286].log_data[18].valid := 1, [1286].log_data[19].valid := 1, [1286].time.Year := 2023, [1286].time.Month := 1, [1286].time.Day := 14, [1286].time.Hour := 3, [1286].time.Minute := 34, [1286].time.Second := 59, [1287].log_data[0].min := 1.0, [1287].log_data[0].max := 1.0, [1287].log_data[0].total := 300.0, [1287].log_data[0].time := 300.0, [1287].log_data[0].minminute := 35, [1287].log_data[0].maxminute := 35, [1287].log_data[0].valid := 1, [1287].log_data[1].valid := 1, [1287].log_data[2].valid := 1, [1287].log_data[3].valid := 1, [1287].log_data[4].valid := 1, [1287].log_data[5].valid := 1,
        [1287].log_data[6].valid := 1, [1287].log_data[7].valid := 1, [1287].log_data[8].valid := 1, [1287].log_data[9].valid := 1, [1287].log_data[10].valid := 1, [1287].log_data[11].valid := 1, [1287].log_data[12].valid := 1, [1287].log_data[13].valid := 1, [1287].log_data[14].valid := 1, [1287].log_data[15].valid := 1, [1287].log_data[16].valid := 1, [1287].log_data[17].valid := 1, [1287].log_data[18].valid := 1, [1287].log_data[19].valid := 1, [1287].time.Year := 2023, [1287].time.Month := 1, [1287].time.Day := 14, [1287].time.Hour := 3, [1287].time.Minute := 39, [1287].time.Second := 59, [1288].log_data[0].min := 1.0, [1288].log_data[0].max := 1.0, [1288].log_data[0].total := 300.0, [1288].log_data[0].time := 300.0, [1288].log_data[0].minminute := 40, [1288].log_data[0].maxminute := 40, [1288].log_data[0].valid := 1, [1288].log_data[1].valid := 1, [1288].log_data[2].valid := 1, [1288].log_data[3].valid := 1, [1288].log_data[4].valid := 1, [1288].log_data[5].valid := 1, [1288].log_data[6].valid := 1, [1288].log_data[7].valid := 1, [1288].log_data[8].valid := 1, [1288].log_data[9].valid := 1, [1288].log_data[10].valid := 1, [1288].log_data[11].valid := 1, [1288].log_data[12].valid := 1, [1288].log_data[13].valid := 1, [1288].log_data[14].valid := 1, [1288].log_data[15].valid := 1, [1288].log_data[16].valid := 1, [1288].log_data[17].valid := 1, [1288].log_data[18].valid := 1, [1288].log_data[19].valid := 1, [1288].time.Year := 2023, [1288].time.Month := 1, [1288].time.Day := 14, [1288].time.Hour := 3, [1288].time.Minute := 44, [1288].time.Second := 59, [1289].log_data[0].min := 1.0, [1289].log_data[0].max := 1.0, [1289].log_data[0].total := 300.0, [1289].log_data[0].time := 300.0, [1289].log_data[0].minminute := 45, [1289].log_data[0].maxminute := 45, [1289].log_data[0].valid := 1, [1289].log_data[1].valid := 1,
        [1289].log_data[2].valid := 1, [1289].log_data[3].valid := 1, [1289].log_data[4].valid := 1, [1289].log_data[5].valid := 1, [1289].log_data[6].valid := 1, [1289].log_data[7].valid := 1, [1289].log_data[8].valid := 1, [1289].log_data[9].valid := 1, [1289].log_data[10].valid := 1, [1289].log_data[11].valid := 1, [1289].log_data[12].valid := 1, [1289].log_data[13].valid := 1, [1289].log_data[14].valid := 1, [1289].log_data[15].valid := 1, [1289].log_data[16].valid := 1, [1289].log_data[17].valid := 1, [1289].log_data[18].valid := 1, [1289].log_data[19].valid := 1, [1289].time.Year := 2023, [1289].time.Month := 1, [1289].time.Day := 14, [1289].time.Hour := 3, [1289].time.Minute := 49, [1289].time.Second := 59, [1290].log_data[0].min := 1.0, [1290].log_data[0].max := 1.0, [1290].log_data[0].total := 300.0, [1290].log_data[0].time := 300.0, [1290].log_data[0].minminute := 50, [1290].log_data[0].maxminute := 50, [1290].log_data[0].valid := 1, [1290].log_data[1].valid := 1, [1290].log_data[2].valid := 1, [1290].log_data[3].valid := 1, [1290].log_data[4].valid := 1, [1290].log_data[5].valid := 1, [1290].log_data[6].valid := 1, [1290].log_data[7].valid := 1, [1290].log_data[8].valid := 1, [1290].log_data[9].valid := 1, [1290].log_data[10].valid := 1, [1290].log_data[11].valid := 1, [1290].log_data[12].valid := 1, [1290].log_data[13].valid := 1, [1290].log_data[14].valid := 1, [1290].log_data[15].valid := 1, [1290].log_data[16].valid := 1, [1290].log_data[17].valid := 1, [1290].log_data[18].valid := 1, [1290].log_data[19].valid := 1, [1290].time.Year := 2023, [1290].time.Month := 1, [1290].time.Day := 14, [1290].time.Hour := 3, [1290].time.Minute := 54, [1290].time.Second := 59, [1291].log_data[0].min := 1.0, [1291].log_data[0].max := 1.0, [1291].log_data[0].total := 300.0, [1291].log_data[0].time := 300.0,
        [1291].log_data[0].minminute := 55, [1291].log_data[0].maxminute := 55, [1291].log_data[0].valid := 1, [1291].log_data[1].valid := 1, [1291].log_data[2].valid := 1, [1291].log_data[3].valid := 1, [1291].log_data[4].valid := 1, [1291].log_data[5].valid := 1, [1291].log_data[6].valid := 1, [1291].log_data[7].valid := 1, [1291].log_data[8].valid := 1, [1291].log_data[9].valid := 1, [1291].log_data[10].valid := 1, [1291].log_data[11].valid := 1, [1291].log_data[12].valid := 1, [1291].log_data[13].valid := 1, [1291].log_data[14].valid := 1, [1291].log_data[15].valid := 1, [1291].log_data[16].valid := 1, [1291].log_data[17].valid := 1, [1291].log_data[18].valid := 1, [1291].log_data[19].valid := 1, [1291].time.Year := 2023, [1291].time.Month := 1, [1291].time.Day := 14, [1291].time.Hour := 3, [1291].time.Minute := 59, [1291].time.Second := 59, [1292].log_data[0].min := 1.0, [1292].log_data[0].max := 1.0, [1292].log_data[0].total := 300.0, [1292].log_data[0].time := 300.0, [1292].log_data[0].valid := 1, [1292].log_data[1].valid := 1, [1292].log_data[2].valid := 1, [1292].log_data[3].valid := 1, [1292].log_data[4].valid := 1, [1292].log_data[5].valid := 1, [1292].log_data[6].valid := 1, [1292].log_data[7].valid := 1, [1292].log_data[8].valid := 1, [1292].log_data[9].valid := 1, [1292].log_data[10].valid := 1, [1292].log_data[11].valid := 1, [1292].log_data[12].valid := 1, [1292].log_data[13].valid := 1, [1292].log_data[14].valid := 1, [1292].log_data[15].valid := 1, [1292].log_data[16].valid := 1, [1292].log_data[17].valid := 1, [1292].log_data[18].valid := 1, [1292].log_data[19].valid := 1, [1292].time.Year := 2023, [1292].time.Month := 1, [1292].time.Day := 14, [1292].time.Hour := 4, [1292].time.Minute := 4, [1292].time.Second := 59, [1293].log_data[0].min := 1.0, [1293].log_data[0].max := 1.0,
        [1293].log_data[0].total := 300.0, [1293].log_data[0].time := 300.0, [1293].log_data[0].minminute := 5, [1293].log_data[0].maxminute := 5, [1293].log_data[0].valid := 1, [1293].log_data[1].valid := 1, [1293].log_data[2].valid := 1, [1293].log_data[3].valid := 1, [1293].log_data[4].valid := 1, [1293].log_data[5].valid := 1, [1293].log_data[6].valid := 1, [1293].log_data[7].valid := 1, [1293].log_data[8].valid := 1, [1293].log_data[9].valid := 1, [1293].log_data[10].valid := 1, [1293].log_data[11].valid := 1, [1293].log_data[12].valid := 1, [1293].log_data[13].valid := 1, [1293].log_data[14].valid := 1, [1293].log_data[15].valid := 1, [1293].log_data[16].valid := 1, [1293].log_data[17].valid := 1, [1293].log_data[18].valid := 1, [1293].log_data[19].valid := 1, [1293].time.Year := 2023, [1293].time.Month := 1, [1293].time.Day := 14, [1293].time.Hour := 4, [1293].time.Minute := 9, [1293].time.Second := 59, [1294].log_data[0].min := 1.0, [1294].log_data[0].max := 1.0, [1294].log_data[0].total := 300.0, [1294].log_data[0].time := 300.0, [1294].log_data[0].minminute := 10, [1294].log_data[0].maxminute := 10, [1294].log_data[0].valid := 1, [1294].log_data[1].valid := 1, [1294].log_data[2].valid := 1, [1294].log_data[3].valid := 1, [1294].log_data[4].valid := 1, [1294].log_data[5].valid := 1, [1294].log_data[6].valid := 1, [1294].log_data[7].valid := 1, [1294].log_data[8].valid := 1, [1294].log_data[9].valid := 1, [1294].log_data[10].valid := 1, [1294].log_data[11].valid := 1, [1294].log_data[12].valid := 1, [1294].log_data[13].valid := 1, [1294].log_data[14].valid := 1, [1294].log_data[15].valid := 1, [1294].log_data[16].valid := 1, [1294].log_data[17].valid := 1, [1294].log_data[18].valid := 1, [1294].log_data[19].valid := 1, [1294].time.Year := 2023, [1294].time.Month := 1, [1294].time.Day := 14, [1294].time.Hour := 4,
        [1294].time.Minute := 14, [1294].time.Second := 59, [1295].log_data[0].min := 1.0, [1295].log_data[0].max := 1.0, [1295].log_data[0].total := 300.0, [1295].log_data[0].time := 300.0, [1295].log_data[0].minminute := 15, [1295].log_data[0].maxminute := 15, [1295].log_data[0].valid := 1, [1295].log_data[1].valid := 1, [1295].log_data[2].valid := 1, [1295].log_data[3].valid := 1, [1295].log_data[4].valid := 1, [1295].log_data[5].valid := 1, [1295].log_data[6].valid := 1, [1295].log_data[7].valid := 1, [1295].log_data[8].valid := 1, [1295].log_data[9].valid := 1, [1295].log_data[10].valid := 1, [1295].log_data[11].valid := 1, [1295].log_data[12].valid := 1, [1295].log_data[13].valid := 1, [1295].log_data[14].valid := 1, [1295].log_data[15].valid := 1, [1295].log_data[16].valid := 1, [1295].log_data[17].valid := 1, [1295].log_data[18].valid := 1, [1295].log_data[19].valid := 1, [1295].time.Year := 2023, [1295].time.Month := 1, [1295].time.Day := 14, [1295].time.Hour := 4, [1295].time.Minute := 19, [1295].time.Second := 59, [1296].log_data[0].min := 1.0, [1296].log_data[0].max := 1.0, [1296].log_data[0].total := 300.0, [1296].log_data[0].time := 300.0, [1296].log_data[0].minminute := 20, [1296].log_data[0].maxminute := 20, [1296].log_data[0].valid := 1, [1296].log_data[1].valid := 1, [1296].log_data[2].valid := 1, [1296].log_data[3].valid := 1, [1296].log_data[4].valid := 1, [1296].log_data[5].valid := 1, [1296].log_data[6].valid := 1, [1296].log_data[7].valid := 1, [1296].log_data[8].valid := 1, [1296].log_data[9].valid := 1, [1296].log_data[10].valid := 1, [1296].log_data[11].valid := 1, [1296].log_data[12].valid := 1, [1296].log_data[13].valid := 1, [1296].log_data[14].valid := 1, [1296].log_data[15].valid := 1, [1296].log_data[16].valid := 1, [1296].log_data[17].valid := 1, [1296].log_data[18].valid := 1, [1296].log_data[19].valid := 1,
        [1296].time.Year := 2023, [1296].time.Month := 1, [1296].time.Day := 14, [1296].time.Hour := 4, [1296].time.Minute := 24, [1296].time.Second := 59, [1297].log_data[0].min := 1.0, [1297].log_data[0].max := 1.0, [1297].log_data[0].total := 300.0, [1297].log_data[0].time := 300.0, [1297].log_data[0].minminute := 25, [1297].log_data[0].maxminute := 25, [1297].log_data[0].valid := 1, [1297].log_data[1].valid := 1, [1297].log_data[2].valid := 1, [1297].log_data[3].valid := 1, [1297].log_data[4].valid := 1, [1297].log_data[5].valid := 1, [1297].log_data[6].valid := 1, [1297].log_data[7].valid := 1, [1297].log_data[8].valid := 1, [1297].log_data[9].valid := 1, [1297].log_data[10].valid := 1, [1297].log_data[11].valid := 1, [1297].log_data[12].valid := 1, [1297].log_data[13].valid := 1, [1297].log_data[14].valid := 1, [1297].log_data[15].valid := 1, [1297].log_data[16].valid := 1, [1297].log_data[17].valid := 1, [1297].log_data[18].valid := 1, [1297].log_data[19].valid := 1, [1297].time.Year := 2023, [1297].time.Month := 1, [1297].time.Day := 14, [1297].time.Hour := 4, [1297].time.Minute := 29, [1297].time.Second := 59, [1298].log_data[0].min := 1.0, [1298].log_data[0].max := 1.0, [1298].log_data[0].total := 300.0, [1298].log_data[0].time := 300.0, [1298].log_data[0].minminute := 30, [1298].log_data[0].maxminute := 30, [1298].log_data[0].valid := 1, [1298].log_data[1].valid := 1, [1298].log_data[2].valid := 1, [1298].log_data[3].valid := 1, [1298].log_data[4].valid := 1, [1298].log_data[5].valid := 1, [1298].log_data[6].valid := 1, [1298].log_data[7].valid := 1, [1298].log_data[8].valid := 1, [1298].log_data[9].valid := 1, [1298].log_data[10].valid := 1, [1298].log_data[11].valid := 1, [1298].log_data[12].valid := 1, [1298].log_data[13].valid := 1, [1298].log_data[14].valid := 1, [1298].log_data[15].valid := 1,
        [1298].log_data[16].valid := 1, [1298].log_data[17].valid := 1, [1298].log_data[18].valid := 1, [1298].log_data[19].valid := 1, [1298].time.Year := 2023, [1298].time.Month := 1, [1298].time.Day := 14, [1298].time.Hour := 4, [1298].time.Minute := 34, [1298].time.Second := 59, [1299].log_data[0].min := 1.0, [1299].log_data[0].max := 1.0, [1299].log_data[0].total := 300.0, [1299].log_data[0].time := 300.0, [1299].log_data[0].minminute := 35, [1299].log_data[0].maxminute := 35, [1299].log_data[0].valid := 1, [1299].log_data[1].valid := 1, [1299].log_data[2].valid := 1, [1299].log_data[3].valid := 1, [1299].log_data[4].valid := 1, [1299].log_data[5].valid := 1, [1299].log_data[6].valid := 1, [1299].log_data[7].valid := 1, [1299].log_data[8].valid := 1, [1299].log_data[9].valid := 1, [1299].log_data[10].valid := 1, [1299].log_data[11].valid := 1, [1299].log_data[12].valid := 1, [1299].log_data[13].valid := 1, [1299].log_data[14].valid := 1, [1299].log_data[15].valid := 1, [1299].log_data[16].valid := 1, [1299].log_data[17].valid := 1, [1299].log_data[18].valid := 1, [1299].log_data[19].valid := 1, [1299].time.Year := 2023, [1299].time.Month := 1, [1299].time.Day := 14, [1299].time.Hour := 4, [1299].time.Minute := 39, [1299].time.Second := 59, [1300].log_data[0].min := 1.0, [1300].log_data[0].max := 1.0, [1300].log_data[0].total := 300.0, [1300].log_data[0].time := 300.0, [1300].log_data[0].minminute := 40, [1300].log_data[0].maxminute := 40, [1300].log_data[0].valid := 1, [1300].log_data[1].valid := 1, [1300].log_data[2].valid := 1, [1300].log_data[3].valid := 1, [1300].log_data[4].valid := 1, [1300].log_data[5].valid := 1, [1300].log_data[6].valid := 1, [1300].log_data[7].valid := 1, [1300].log_data[8].valid := 1, [1300].log_data[9].valid := 1, [1300].log_data[10].valid := 1, [1300].log_data[11].valid := 1,
